KUKA KRL program: MyProgram_240().src

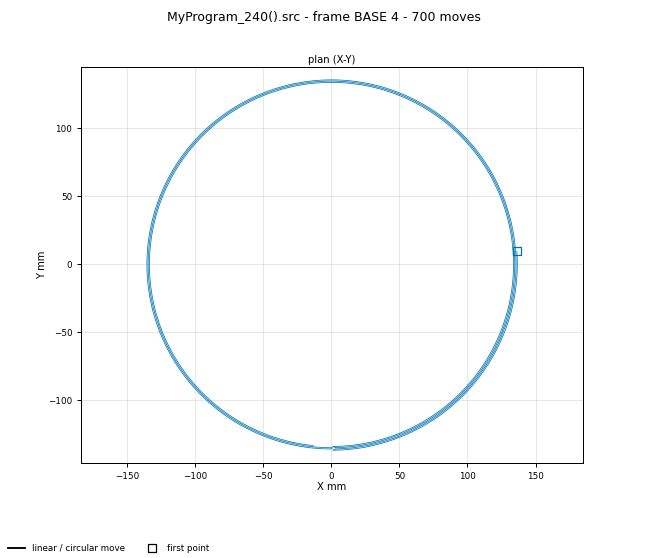
[picture p0: tool path of MyProgram_240().src in frame BASE 4, 700 of 700 moves have a stored position in this frame; points joined in program order, loops and branches not executed]
&ACCESS RVP
&REL 1
&PARAM TEMPLATE = C:\KRC\Roboter\Template\vorgabe
&PARAM EDITMASK = *
DEF MyProgram_240()
; ---- Setting reference (Base) ----
$BASE = BASE_DATA[4]

; --------------------------
; ---- Setting tool (TCP) ----
$TOOL = TOOL_DATA[3]
; --------------------------

$VEL.CP = VEL_APROX_PRINT
Startdeposition()
$VEL.CP = VEL_PRINT
LIN {X 136.2773,Y 9.5637,Z 161,A 0.3979,B 23.0272,C -1.0447,E1 23.2091,E2 806.9336} C_DIS
LIN {X 136.5182,Y 5.0682,Z 161,A -1.0464,B 23.0264,C -1.0618,E1 23.2093,E2 808.325} C_DIS
LIN {X 136.6137,Y -0.1543,Z 161,A -3.2724,B 23.0268,C -1.0528,E1 23.2093,E2 810.5594} C_DIS
LIN {X 136.5514,Y -4.0769,Z 161,A -4.8375,B 23.0268,C -1.0517,E1 23.2093,E2 812.1172} C_DIS
LIN {X 136.345,Y -8.5376,Z 161,A -6.6605,B 23.027,C -1.0482,E1 23.209,E2 813.9371} C_DIS
LIN {X 136.0456,Y -12.4414,Z 161,A -8.3456,B 23.0274,C -1.0406,E1 23.2086,E2 815.6307} C_DIS
LIN {X 135.6641,Y -16.0648,Z 161,A -10.3586,B 23.0286,C -1.0102,E1 23.2079,E2 817.7078} C_DIS
LIN {X 135.0038,Y -20.8989,Z 161,A -11.8021,B 23.0276,C -1.0351,E1 23.2074,E2 819.0787} C_DIS
LIN {X 134.4014,Y -24.4787,Z 161,A -13.4389,B 23.0281,C -1.0242,E1 23.2066,E2 820.7328} C_DIS
LIN {X 133.5686,Y -28.6745,Z 161,A -15.1069,B 23.0281,C -1.025,E1 23.2056,E2 822.388} C_DIS
LIN {X 132.7943,Y -32.0691,Z 161,A -16.5169,B 23.0281,C -1.023,E1 23.2047,E2 823.7942} C_DIS
LIN {X 131.9632,Y -35.3339,Z 161,A -17.9644,B 23.0284,C -1.0166,E1 23.2037,E2 825.2487} C_DIS
LIN {X 130.9854,Y -38.8039,Z 161,A -19.4634,B 23.0285,C -1.0125,E1 23.2025,E2 826.7489} C_DIS
LIN {X 129.5513,Y -43.3501,Z 161,A -21.4628,B 23.0288,C -1.0062,E1 23.2008,E2 828.7519} C_DIS
LIN {X 128.1195,Y -47.4171,Z 161,A -23.8257,B 23.0302,C -0.9715,E1 23.1985,E2 831.1885} C_DIS
LIN {X 126.3141,Y -52.0373,Z 161,A -25.224,B 23.029,C -1.0007,E1 23.1971,E2 832.504} C_DIS
LIN {X 124.3025,Y -56.6756,Z 161,A -27.3549,B 23.0293,C -0.9937,E1 23.1947,E2 834.6401} C_DIS
LIN {X 123.0552,Y -59.3326,Z 161,A -28.6015,B 23.0295,C -0.9891,E1 23.1932,E2 835.8908} C_DIS
LIN {X 121.4701,Y -62.5145,Z 161,A -30.119,B 23.0297,C -0.9833,E1 23.1913,E2 837.4144} C_DIS
LIN {X 119.0587,Y -66.9945,Z 161,A -32.2949,B 23.0301,C -0.9747,E1 23.1884,E2 839.5996} C_DIS
LIN {X 116.8471,Y -70.7814,Z 161,A -34.3743,B 23.0308,C -0.9568,E1 23.1853,E2 841.7128} C_DIS
LIN {X 115.0222,Y -73.7098,Z 161,A -35.319,B 23.0299,C -0.979,E1 23.184,E2 842.596} C_DIS
LIN {X 112.7004,Y -77.2131,Z 161,A -37.1335,B 23.0302,C -0.9713,E1 23.1812,E2 844.4202} C_DIS
LIN {X 110.946,Y -79.7139,Z 161,A -38.6151,B 23.0308,C -0.9572,E1 23.1788,E2 845.9297} C_DIS
LIN {X 108.2978,Y -83.2762,Z 161,A -40.4743,B 23.031,C -0.9523,E1 23.1756,E2 847.7917} C_DIS
LIN {X 105.5105,Y -86.7809,Z 161,A -42.2839,B 23.031,C -0.9508,E1 23.1724,E2 849.5958} C_DIS
LIN {X 102.8746,Y -89.8891,Z 161,A -44.0205,B 23.0313,C -0.945,E1 23.1693,E2 851.3386} C_DIS
LIN {X 100.0782,Y -92.9925,Z 161,A -45.7792,B 23.0314,C -0.9401,E1 23.166,E2 853.1011} C_DIS
LIN {X 96.8908,Y -96.3089,Z 161,A -47.6911,B 23.0316,C -0.9363,E1 23.1622,E2 855.0138} C_DIS
LIN {X 93.7473,Y -99.3714,Z 161,A -49.4881,B 23.0316,C -0.9341,E1 23.1586,E2 856.8082} C_DIS
LIN {X 90.5239,Y -102.3164,Z 161,A -51.3153,B 23.0318,C -0.93,E1 23.1548,E2 858.6377} C_DIS
LIN {X 87.2594,Y -105.1145,Z 161,A -53.1447,B 23.032,C -0.9246,E1 23.1509,E2 860.4732} C_DIS
LIN {X 83.7135,Y -107.9596,Z 161,A -55.0296,B 23.0322,C -0.9216,E1 23.1468,E2 862.3582} C_DIS
LIN {X 79.9438,Y -110.7803,Z 161,A -56.981,B 23.0322,C -0.9186,E1 23.1424,E2 864.3095} C_DIS
LIN {X 76.3648,Y -113.2771,Z 161,A -58.824,B 23.0324,C -0.9142,E1 23.1381,E2 866.1567} C_DIS
LIN {X 72.5813,Y -115.7382,Z 161,A -60.7513,B 23.0326,C -0.9088,E1 23.1336,E2 868.0909} C_DIS
LIN {X 68.7664,Y -118.0447,Z 161,A -62.5822,B 23.0326,C -0.9074,E1 23.1292,E2 869.9194} C_DIS
LIN {X 64.8661,Y -120.2317,Z 161,A -64.9487,B 23.0337,C -0.879,E1 23.1232,E2 872.3506} C_DIS
LIN {X 60.5233,Y -122.4729,Z 161,A -66.0976,B 23.0322,C -0.9217,E1 23.1207,E2 873.3874} C_DIS
LIN {X 58.242,Y -123.5762,Z 161,A -67.4262,B 23.0327,C -0.9063,E1 23.1172,E2 874.7514} C_DIS
LIN {X 54.9164,Y -125.0898,Z 161,A -69.3172,B 23.0335,C -0.8857,E1 23.1122,E2 876.6899} C_DIS
LIN {X 51.6442,Y -126.4751,Z 161,A -70.416,B 23.0328,C -0.9034,E1 23.1095,E2 877.7406} C_DIS
LIN {X 45.2029,Y -128.9172,Z 161,A -73.1919,B 23.0328,C -0.9053,E1 23.1023,E2 880.5052} C_DIS
LIN {X 41.5898,Y -130.1269,Z 161,A -74.9321,B 23.0331,C -0.8961,E1 23.0976,E2 882.2652} C_DIS
LIN {X 36.528,Y -131.6378,Z 161,A -77.0528,B 23.0331,C -0.8984,E1 23.092,E2 884.3759} C_DIS
LIN {X 33.7209,Y -132.3845,Z 161,A -78.3762,B 23.0333,C -0.8919,E1 23.0884,E2 885.714} C_DIS
LIN {X 30.5077,Y -133.1617,Z 161,A -79.7785,B 23.0333,C -0.8897,E1 23.0845,E2 887.1194} C_DIS
LIN {X 26.5179,Y -134.0153,Z 161,A -81.6868,B 23.0338,C -0.8783,E1 23.0792,E2 889.0544} C_DIS
LIN {X 22.9609,Y -134.6693,Z 161,A -82.9925,B 23.0334,C -0.8877,E1 23.0757,E2 890.3344} C_DIS
LIN {X 19.4058,Y -135.2265,Z 161,A -84.8817,B 23.0341,C -0.8677,E1 23.0704,E2 892.2729} C_DIS
LIN {X 15.342,Y -135.7496,Z 161,A -86.2543,B 23.0336,C -0.8839,E1 23.0667,E2 893.6031} C_DIS
LIN {X 8.2701,Y -136.3615,Z 161,A -89.1847,B 23.0336,C -0.8848,E1 23.0585,E2 896.5294} C_DIS
LIN {X 0.9864,Y -136.6083,Z 161,A -93.055,B 23.035,C -0.8438,E1 23.0474,E2 900.5038} C_DIS
Enddeposition()
LIN {X 0.9864,Y -136.6083,Z 161,A -93.055,B 23.035,C -0.8438,E1 23.0474,E2 900.5038} C_DIS
Startdeposition()
$VEL.CP = VEL_PRINT
LIN {X 2.6306,Y -135.6628,Z 161,A -90.3615,B 21.7658,C -0.7295,E1 21.7824,E2 897.9751} C_DIS
LIN {X 6.721,Y -135.5212,Z 161,A -88.7348,B 21.766,C -0.7253,E1 21.7869,E2 896.3603} C_DIS
LIN {X 9.445,Y -135.3593,Z 161,A -87.4479,B 21.7658,C -0.7322,E1 21.7905,E2 895.0556} C_DIS
LIN {X 14.134,Y -134.9501,Z 161,A -85.5629,B 21.7658,C -0.7283,E1 21.7957,E2 893.1824} C_DIS
LIN {X 18.0786,Y -134.4786,Z 161,A -83.8012,B 21.7658,C -0.7334,E1 21.8006,E2 891.4087} C_DIS
LIN {X 22.3172,Y -133.8397,Z 161,A -82.1872,B 21.766,C -0.7253,E1 21.805,E2 889.8183} C_DIS
LIN {X 24.8651,Y -133.3913,Z 161,A -80.9711,B 21.7658,C -0.732,E1 21.8084,E2 888.5856} C_DIS
LIN {X 28.3569,Y -132.6916,Z 161,A -79.5518,B 21.7658,C -0.7293,E1 21.8122,E2 887.1758} C_DIS
LIN {X 31.5596,Y -131.9665,Z 161,A -78.1631,B 21.7658,C -0.7307,E1 21.816,E2 885.7857} C_DIS
LIN {X 34.2506,Y -131.2956,Z 161,A -76.8928,B 21.7656,C -0.7366,E1 21.8195,E2 884.5017} C_DIS
LIN {X 40.5935,Y -129.4745,Z 161,A -74.0549,B 21.7654,C -0.7422,E1 21.8271,E2 881.6545} C_DIS
LIN {X 44.4809,Y -128.1894,Z 161,A -72.4077,B 21.7654,C -0.7404,E1 21.8314,E2 880.016} C_DIS
LIN {X 48.4743,Y -126.7353,Z 161,A -70.6142,B 21.7654,C -0.7426,E1 21.8361,E2 878.2208} C_DIS
LIN {X 52.0834,Y -125.2933,Z 161,A -68.9248,B 21.7653,C -0.7473,E1 21.8405,E2 876.5234} C_DIS
LIN {X 56.601,Y -123.3187,Z 161,A -67.1132,B 21.7656,C -0.7373,E1 21.8451,E2 874.7439} C_DIS
LIN {X 60.0155,Y -121.6929,Z 161,A -64.3194,B 21.7635,C -0.7986,E1 21.8525,E2 871.7941} C_DIS
LIN {X 66.7124,Y -118.157,Z 161,A -62.0959,B 21.765,C -0.756,E1 21.8576,E2 869.6927} C_DIS
LIN {X 72.0742,Y -114.9654,Z 161,A -59.4888,B 21.7649,C -0.7595,E1 21.8638,E2 867.0857} C_DIS
LIN {X 75.5582,Y -112.7058,Z 161,A -57.7533,B 21.7648,C -0.762,E1 21.8679,E2 865.3501} C_DIS
LIN {X 79.2761,Y -110.1229,Z 161,A -55.828,B 21.7646,C -0.7665,E1 21.8722,E2 863.4205} C_DIS
LIN {X 82.83,Y -107.4751,Z 161,A -53.9837,B 21.7646,C -0.7692,E1 21.8763,E2 861.577} C_DIS
LIN {X 86.0296,Y -104.931,Z 161,A -52.2698,B 21.7644,C -0.7723,E1 21.8801,E2 859.8621} C_DIS
LIN {X 89.4999,Y -101.9876,Z 161,A -50.3307,B 21.7643,C -0.7775,E1 21.8842,E2 857.918} C_DIS
LIN {X 92.7399,Y -99.0506,Z 161,A -48.5154,B 21.7642,C -0.7803,E1 21.8879,E2 856.1039} C_DIS
LIN {X 95.8163,Y -96.0774,Z 161,A -46.7327,B 21.7641,C -0.7834,E1 21.8915,E2 854.3216} C_DIS
LIN {X 98.8991,Y -92.9011,Z 161,A -44.8508,B 21.7639,C -0.7886,E1 21.8951,E2 852.4351} C_DIS
LIN {X 101.9435,Y -89.5503,Z 161,A -42.9731,B 21.7638,C -0.7918,E1 21.8986,E2 850.5587} C_DIS
LIN {X 104.6052,Y -86.4253,Z 161,A -41.2947,B 21.7638,C -0.7936,E1 21.9016,E2 848.8846} C_DIS
LIN {X 107.2944,Y -83.0631,Z 161,A -39.44,B 21.7635,C -0.8002,E1 21.9048,E2 847.0222} C_DIS
LIN {X 110.0674,Y -79.3526,Z 161,A -37.6745,B 21.7636,C -0.796,E1 21.9077,E2 845.2779} C_DIS
LIN {X 113.15,Y -74.8916,Z 161,A -35.3067,B 21.7633,C -0.8062,E1 21.9115,E2 842.8963} C_DIS
LIN {X 116.0911,Y -70.2454,Z 161,A -32.9144,B 21.7629,C -0.8163,E1 21.915,E2 840.4912} C_DIS
LIN {X 117.6865,Y -67.5395,Z 161,A -31.2671,B 21.7622,C -0.8362,E1 21.9174,E2 838.8005} C_DIS
LIN {X 119.6001,Y -64.089,Z 161,A -29.8843,B 21.7625,C -0.8268,E1 21.9191,E2 837.4512} C_DIS
LIN {X 121.5521,Y -60.301,Z 161,A -28.2528,B 21.7626,C -0.8238,E1 21.9212,E2 835.8381} C_DIS
LIN {X 122.9704,Y -57.3542,Z 161,A -27.0274,B 21.7628,C -0.8201,E1 21.9226,E2 834.63} C_DIS
LIN {X 124.2951,Y -54.4258,Z 161,A -25.4063,B 21.7621,C -0.8374,E1 21.9245,E2 832.973} C_DIS
LIN {X 127.902,Y -45.3069,Z 161,A -21.4308,B 21.762,C -0.8417,E1 21.9285,E2 829.0118} C_DIS
LIN {X 129.6738,Y -39.9479,Z 161,A -19.1656,B 21.762,C -0.8432,E1 21.9304,E2 826.7574} C_DIS
LIN {X 130.6686,Y -36.5623,Z 161,A -17.5786,B 21.7616,C -0.8527,E1 21.9317,E2 825.1555} C_DIS
LIN {X 131.5001,Y -33.4486,Z 161,A -16.2258,B 21.7614,C -0.8566,E1 21.9326,E2 823.8013} C_DIS
LIN {X 132.3825,Y -29.7689,Z 161,A -14.5067,B 21.761,C -0.8678,E1 21.9337,E2 822.064} C_DIS
LIN {X 133.3015,Y -25.3348,Z 161,A -12.6917,B 21.761,C -0.869,E1 21.9347,E2 820.2581} C_DIS
LIN {X 134.0395,Y -21.0869,Z 161,A -11.1256,B 21.7612,C -0.8621,E1 21.9354,E2 818.7212} C_DIS
LIN {X 134.4989,Y -17.9238,Z 161,A -9.451,B 21.7604,C -0.8827,E1 21.9361,E2 817.003} C_DIS
LIN {X 135.0397,Y -13.2483,Z 161,A -7.7651,B 21.7608,C -0.8739,E1 21.9366,E2 815.3521} C_DIS
LIN {X 135.317,Y -10.025,Z 161,A -6.2881,B 21.7604,C -0.8839,E1 21.9369,E2 813.8587} C_DIS
LIN {X 135.5188,Y -6.7689,Z 161,A -4.8555,B 21.7601,C -0.8911,E1 21.9371,E2 812.4167} C_DIS
LIN {X 135.6615,Y -2.7083,Z 161,A -3.0725,B 21.7598,C -0.9,E1 21.9372,E2 810.6223} C_DIS
LIN {X 135.6756,Y 1.8649,Z 161,A -1.2349,B 21.7598,C -0.9015,E1 21.9372,E2 808.7933} C_DIS
LIN {X 135.5773,Y 5.478,Z 161,A 0.0506,B 21.76,C -0.8943,E1 21.9372,E2 807.5359} C_DIS
LIN {X 135.424,Y 8.4577,Z 161,A 1.4958,B 21.7595,C -0.9076,E1 21.9369,E2 806.0652} C_DIS
LIN {X 135.1194,Y 12.4177,Z 161,A 3.254,B 21.7591,C -0.917,E1 21.9365,E2 804.2939} C_DIS
LIN {X 134.6789,Y 16.5206,Z 161,A 5.014,B 21.7588,C -0.9234,E1 21.9359,E2 802.5289} C_DIS
LIN {X 134.157,Y 20.3276,Z 161,A 6.5505,B 21.7588,C -0.9242,E1 21.9353,E2 801.0008} C_DIS
LIN {X 133.5954,Y 23.7364,Z 161,A 7.9477,B 21.7588,C -0.9257,E1 21.9346,E2 799.6092} C_DIS
LIN {X 132.9372,Y 27.1812,Z 161,A 9.4648,B 21.7585,C -0.9322,E1 21.9338,E2 798.0852} C_DIS
LIN {X 131.9188,Y 31.7572,Z 161,A 11.3888,B 21.7583,C -0.9355,E1 21.9326,E2 796.1652} C_DIS
LIN {X 130.9966,Y 35.3717,Z 161,A 13.0456,B 21.758,C -0.9444,E1 21.9314,E2 794.4958} C_DIS
LIN {X 127.8094,Y 45.5637,Z 161,A 17.4828,B 21.7576,C -0.9542,E1 21.9276,E2 790.0616} C_DIS
LIN {X 125.7762,Y 50.9062,Z 161,A 19.7346,B 21.7576,C -0.9532,E1 21.9254,E2 787.8269} C_DIS
LIN {X 124.6706,Y 53.5573,Z 161,A 21.0157,B 21.7573,C -0.9601,E1 21.9239,E2 786.5356} C_DIS
LIN {X 123.2293,Y 56.7944,Z 161,A 22.3641,B 21.7574,C -0.9571,E1 21.9224,E2 785.2039} C_DIS
LIN {X 121.8558,Y 59.6853,Z 161,A 23.906,B 21.7569,C -0.9703,E1 21.9205,E2 783.6363} C_DIS
LIN {X 120.1715,Y 63.0066,Z 161,A 25.3923,B 21.7569,C -0.9703,E1 21.9186,E2 782.1589} C_DIS
LIN {X 118.0968,Y 66.8196,Z 161,A 27.3535,B 21.7564,C -0.9817,E1 21.9159,E2 780.1793} C_DIS
LIN {X 115.9673,Y 70.4502,Z 161,A 29.0848,B 21.7564,C -0.9841,E1 21.9135,E2 778.4518} C_DIS
LIN {X 113.606,Y 74.1983,Z 161,A 30.9425,B 21.7561,C -0.9884,E1 21.9107,E2 776.5935} C_DIS
LIN {X 111.8562,Y 76.8098,Z 161,A 32.7606,B 21.7549,C -1.016,E1 21.9077,E2 774.7118} C_DIS
LIN {X 109.0292,Y 80.7731,Z 161,A 34.3198,B 21.7558,C -0.9966,E1 21.9052,E2 773.2134} C_DIS
LIN {X 105.9568,Y 84.7633,Z 161,A 36.4456,B 21.7555,C -1.0017,E1 21.9015,E2 771.0856} C_DIS
LIN {X 103.0638,Y 88.2586,Z 161,A 38.231,B 21.7556,C -0.9998,E1 21.8983,E2 769.3149} C_DIS
LIN {X 99.7809,Y 91.9528,Z 161,A 40.3381,B 21.7554,C -1.0055,E1 21.8944,E2 767.2033} C_DIS
LIN {X 96.9434,Y 94.9397,Z 161,A 42.1274,B 21.7551,C -1.0117,E1 21.8909,E2 765.4063} C_DIS
LIN {X 94.8714,Y 97.0104,Z 161,A 43.4385,B 21.7548,C -1.018,E1 21.8883,E2 764.0849} C_DIS
LIN {X 91.3906,Y 100.2966,Z 161,A 45.411,B 21.7548,C -1.0197,E1 21.8843,E2 762.117} C_DIS
LIN {X 88.4188,Y 102.9257,Z 161,A 48.0168,B 21.7525,C -1.0685,E1 21.8785,E2 759.392} C_DIS
LIN {X 82.6709,Y 107.5973,Z 161,A 50.1675,B 21.7544,C -1.0265,E1 21.874,E2 757.3633} C_DIS
LIN {X 78.7472,Y 110.5011,Z 161,A 52.2253,B 21.7543,C -1.03,E1 21.8694,E2 755.3048} C_DIS
LIN {X 75.2259,Y 112.9276,Z 161,A 54.0074,B 21.7542,C -1.0319,E1 21.8652,E2 753.5247} C_DIS
LIN {X 71.3591,Y 115.4105,Z 161,A 55.926,B 21.7542,C -1.0338,E1 21.8607,E2 751.608} C_DIS
LIN {X 67.6548,Y 117.6203,Z 161,A 57.7882,B 21.7539,C -1.0385,E1 21.8562,E2 749.7399} C_DIS
LIN {X 63.7967,Y 119.7566,Z 161,A 59.6822,B 21.7537,C -1.0426,E1 21.8515,E2 747.8413} C_DIS
LIN {X 60.4556,Y 121.4758,Z 161,A 61.1704,B 21.7538,C -1.04,E1 21.8479,E2 746.3649} C_DIS
LIN {X 57.2122,Y 123.0361,Z 161,A 62.6232,B 21.7538,C -1.0386,E1 21.8442,E2 744.92} C_DIS
LIN {X 53.899,Y 124.5229,Z 161,A 64.1049,B 21.7539,C -1.0379,E1 21.8404,E2 743.4443} C_DIS
LIN {X 46.6483,Y 127.4184,Z 161,A 67.3702,B 21.7539,C -1.0397,E1 21.832,E2 740.1828} C_DIS
LIN {X 42.5099,Y 128.857,Z 161,A 69.3414,B 21.7535,C -1.047,E1 21.8267,E2 738.1963} C_DIS
LIN {X 38.5045,Y 130.1101,Z 161,A 71.0992,B 21.7535,C -1.0477,E1 21.822,E2 736.4403} C_DIS
LIN {X 35.0814,Y 131.074,Z 161,A 72.5366,B 21.7535,C -1.0458,E1 21.8182,E2 735.0109} C_DIS
LIN {X 31.831,Y 131.901,Z 161,A 73.8763,B 21.7537,C -1.0431,E1 21.8146,E2 733.6809} C_DIS
LIN {X 28.7421,Y 132.6085,Z 161,A 75.383,B 21.7533,C -1.0517,E1 21.8104,E2 732.1534} C_DIS
LIN {X 24.7943,Y 133.4048,Z 161,A 76.9366,B 21.7536,C -1.0455,E1 21.8062,E2 730.6184} C_DIS
LIN {X 20.8451,Y 134.0769,Z 161,A 78.478,B 21.7539,C -1.0392,E1 21.802,E2 729.096} C_DIS
LIN {X 18.6136,Y 134.4061,Z 161,A 79.7449,B 21.7532,C -1.054,E1 21.7984,E2 727.7904} C_DIS
LIN {X 14.7979,Y 134.8786,Z 161,A 81.3068,B 21.7532,C -1.0515,E1 21.7941,E2 726.2366} C_DIS
LIN {X 11.9597,Y 135.1607,Z 161,A 82.5203,B 21.7532,C -1.0521,E1 21.7907,E2 725.0224} C_DIS
LIN {X 7.7951,Y 135.4648,Z 161,A 84.3117,B 21.7532,C -1.0535,E1 21.7857,E2 723.2282} C_DIS
LIN {X 3.449,Y 135.6443,Z 161,A 86.2031,B 21.7531,C -1.0559,E1 21.7804,E2 721.3308} C_DIS
LIN {X -0.0735,Y 135.6895,Z 161,A 87.6782,B 21.7531,C -1.0551,E1 21.7763,E2 719.858} C_DIS
LIN {X -4.1066,Y 135.6261,Z 161,A 89.3542,B 21.7532,C -1.0534,E1 21.7716,E2 718.1863} C_DIS
LIN {X -8.3893,Y 135.4282,Z 161,A 91.1318,B 21.7533,C -1.0513,E1 21.7667,E2 716.4138} C_DIS
LIN {X -12.9086,Y 135.0723,Z 161,A 92.8361,B 21.7538,C -1.0409,E1 21.762,E2 714.7366} C_DIS
LIN {X -15.9106,Y 134.7517,Z 161,A 94.0719,B 21.7538,C -1.0385,E1 21.7586,E2 713.5065} C_DIS
LIN {X -19.1715,Y 134.3264,Z 161,A 95.6577,B 21.7535,C -1.0466,E1 21.7542,E2 711.8974} C_DIS
LIN {X -22.7522,Y 133.7671,Z 161,A 97.2253,B 21.7535,C -1.0472,E1 21.7498,E2 710.3264} C_DIS
LIN {X -26.7692,Y 133.0211,Z 161,A 98.8877,B 21.7537,C -1.0431,E1 21.7453,E2 708.6731} C_DIS
LIN {X -30.0117,Y 132.327,Z 161,A 100.3431,B 21.7537,C -1.0444,E1 21.7413,E2 707.212} C_DIS
LIN {X -33.3937,Y 131.5141,Z 161,A 101.8139,B 21.7537,C -1.0431,E1 21.7373,E2 705.7422} C_DIS
LIN {X -41.2355,Y 129.2699,Z 161,A 105.3327,B 21.7537,C -1.0428,E1 21.7279,E2 702.2177} C_DIS
LIN {X -44.9986,Y 128.0099,Z 161,A 107.0495,B 21.7537,C -1.0426,E1 21.7233,E2 700.4975} C_DIS
LIN {X -48.5735,Y 126.6967,Z 161,A 108.4612,B 21.7542,C -1.0317,E1 21.7197,E2 699.1118} C_DIS
LIN {X -51.8102,Y 125.4074,Z 161,A 109.8953,B 21.7544,C -1.0281,E1 21.716,E2 697.6838} C_DIS
LIN {X -54.485,Y 124.2695,Z 161,A 111.3741,B 21.7539,C -1.0375,E1 21.7122,E2 696.1754} C_DIS
LIN {X -58.2306,Y 122.5574,Z 161,A 112.7848,B 21.7547,C -1.0203,E1 21.7087,E2 694.8071} C_DIS
LIN {X -61.2691,Y 121.067,Z 161,A 114.5593,B 21.7541,C -1.0334,E1 21.7042,E2 692.9918} C_DIS
LIN {X -66.3889,Y 118.3389,Z 161,A 117.0044,B 21.7543,C -1.0291,E1 21.6982,E2 690.5503} C_DIS
LIN {X -70.5015,Y 115.9363,Z 161,A 118.9693,B 21.7546,C -1.0234,E1 21.6935,E2 688.5937} C_DIS
LIN {X -74.8528,Y 113.1755,Z 161,A 121.8836,B 21.7533,C -1.0521,E1 21.6865,E2 685.5906} C_DIS
LIN {X -79.6697,Y 109.8376,Z 161,A 123.6709,B 21.7549,C -1.0166,E1 21.6826,E2 683.8922} C_DIS
LIN {X -82.3618,Y 107.8337,Z 161,A 125.4147,B 21.7544,C -1.0281,E1 21.6787,E2 682.11} C_DIS
LIN {X -85.4101,Y 105.4361,Z 161,A 126.7086,B 21.7552,C -1.0095,E1 21.6759,E2 680.8609} C_DIS
LIN {X -88.7115,Y 102.6737,Z 161,A 128.5803,B 21.7552,C -1.0078,E1 21.6719,E2 678.9852} C_DIS
LIN {X -92.1214,Y 99.6261,Z 161,A 130.5442,B 21.7554,C -1.0048,E1 21.6679,E2 677.0201} C_DIS
LIN {X -95.2819,Y 96.6077,Z 161,A 132.3637,B 21.7556,C -0.9994,E1 21.6642,E2 675.2066} C_DIS
LIN {X -98.1476,Y 93.6943,Z 161,A 134.044,B 21.7559,C -0.9932,E1 21.661,E2 673.5345} C_DIS
LIN {X -100.9175,Y 90.7044,Z 161,A 135.8256,B 21.7559,C -0.9916,E1 21.6576,E2 671.7481} C_DIS
LIN {X -105.2895,Y 85.5906,Z 161,A 138.6205,B 21.7564,C -0.9823,E1 21.6526,E2 668.9635} C_DIS
LIN {X -108.6887,Y 81.2305,Z 161,A 141.0706,B 21.7564,C -0.9811,E1 21.6485,E2 666.5029} C_DIS
LIN {X -110.9298,Y 78.1419,Z 161,A 143.0908,B 21.7559,C -0.9945,E1 21.6451,E2 664.4348} C_DIS
LIN {X -113.4209,Y 74.4801,Z 161,A 144.4907,B 21.757,C -0.9689,E1 21.6431,E2 663.0962} C_DIS
LIN {X -115.6634,Y 70.9475,Z 161,A 146.2696,B 21.7571,C -0.9645,E1 21.6404,E2 661.3188} C_DIS
LIN {X -117.6966,Y 67.5217,Z 161,A 147.7352,B 21.7577,C -0.9503,E1 21.6384,E2 659.8827} C_DIS
LIN {X -119.9419,Y 63.4439,Z 161,A 149.8673,B 21.7577,C -0.9518,E1 21.6355,E2 657.7335} C_DIS
LIN {X -121.4837,Y 60.4397,Z 161,A 151.5472,B 21.7574,C -0.9586,E1 21.6334,E2 656.0247} C_DIS
LIN {X -123.6736,Y 55.822,Z 161,A 153.5716,B 21.7579,C -0.9464,E1 21.631,E2 654.0205} C_DIS
LIN {X -125.1307,Y 52.4727,Z 161,A 155.0695,B 21.7582,C -0.9398,E1 21.6294,E2 652.5307} C_DIS
LIN {X -126.2395,Y 49.7498,Z 161,A 156.4219,B 21.7582,C -0.9408,E1 21.628,E2 651.1669} C_DIS
LIN {X -127.5477,Y 46.2895,Z 161,A 157.8668,B 21.7585,C -0.931,E1 21.6266,E2 649.739} C_DIS
LIN {X -128.5417,Y 43.4566,Z 161,A 159.3197,B 21.7584,C -0.935,E1 21.6253,E2 648.2656} C_DIS
LIN {X -129.6308,Y 40.0885,Z 161,A 160.711,B 21.7587,C -0.9259,E1 21.6241,E2 646.8896} C_DIS
LIN {X -130.6087,Y 36.7763,Z 161,A 162.1278,B 21.759,C -0.9196,E1 21.623,E2 645.4805} C_DIS
LIN {X -131.4745,Y 33.5498,Z 161,A 163.5569,B 21.7591,C -0.9159,E1 21.622,E2 644.0515} C_DIS
LIN {X -132.2559,Y 30.3232,Z 161,A 164.9557,B 21.7593,C -0.9114,E1 21.6211,E2 642.6555} C_DIS
LIN {X -132.8535,Y 27.5927,Z 161,A 166.2341,B 21.7593,C -0.9118,E1 21.6204,E2 641.3671} C_DIS
LIN {X -133.507,Y 24.2301,Z 161,A 167.4819,B 21.7598,C -0.8987,E1 21.6197,E2 640.1462} C_DIS
LIN {X -134.0793,Y 20.8299,Z 161,A 169.1016,B 21.7598,C -0.9011,E1 21.619,E2 638.5089} C_DIS
LIN {X -134.5669,Y 17.4053,Z 161,A 170.6261,B 21.7598,C -0.8991,E1 21.6184,E2 636.979} C_DIS
LIN {X -135.0616,Y 13.0198,Z 161,A 172.4817,B 21.76,C -0.8928,E1 21.6179,E2 635.1276} C_DIS
LIN {X -135.4054,Y 8.7594,Z 161,A 174.3182,B 21.7602,C -0.8884,E1 21.6175,E2 633.2902} C_DIS
LIN {X -135.5926,Y 5.0854,Z 161,A 175.8945,B 21.7604,C -0.8844,E1 21.6173,E2 631.7137} C_DIS
LIN {X -135.6855,Y 0.8916,Z 161,A 177.628,B 21.7607,C -0.8771,E1 21.6173,E2 629.9879} C_DIS
LIN {X -135.659,Y -2.862,Z 161,A 179.3405,B 21.7607,C -0.8775,E1 21.6173,E2 628.2622} C_DIS
LIN {X -135.5073,Y -6.9975,Z 161,A -179.0048,B 21.761,C -0.8679,E1 21.6175,E2 626.6218} C_DIS
LIN {X -135.232,Y -11.116,Z 161,A -177.2662,B 21.7612,C -0.8622,E1 21.6179,E2 624.8867} C_DIS
LIN {X -134.9048,Y -14.5547,Z 161,A -175.8003,B 21.7614,C -0.8579,E1 21.6183,E2 623.4221} C_DIS
LIN {X -134.431,Y -18.4399,Z 161,A -174.0261,B 21.7614,C -0.8579,E1 21.6189,E2 621.6356} C_DIS
LIN {X -133.8734,Y -22.1149,Z 161,A -172.55,B 21.7617,C -0.8489,E1 21.6196,E2 620.1735} C_DIS
LIN {X -133.3708,Y -24.9719,Z 161,A -171.4418,B 21.762,C -0.8401,E1 21.6201,E2 619.0817} C_DIS
LIN {X -132.1859,Y -30.6296,Z 161,A -168.7455,B 21.762,C -0.8435,E1 21.6218,E2 616.3575} C_DIS
LIN {X -131.2802,Y -34.3081,Z 161,A -166.9877,B 21.7618,C -0.8454,E1 21.623,E2 614.5824} C_DIS
LIN {X -129.8793,Y -39.2766,Z 161,A -165.0969,B 21.7625,C -0.8263,E1 21.6244,E2 612.7307} C_DIS
LIN {X -129.0208,Y -42.0153,Z 161,A -163.6523,B 21.7623,C -0.8328,E1 21.6257,E2 611.259} C_DIS
LIN {X -127.7402,Y -45.7555,Z 161,A -162.3613,B 21.7631,C -0.8115,E1 21.6268,E2 610.0172} C_DIS
LIN {X -126.632,Y -48.7402,Z 161,A -160.7495,B 21.7628,C -0.8191,E1 21.6284,E2 608.3741} C_DIS
LIN {X -125.2904,Y -52.0903,Z 161,A -159.2589,B 21.763,C -0.8132,E1 21.63,E2 606.8898} C_DIS
LIN {X -124.1683,Y -54.716,Z 161,A -157.4205,B 21.7621,C -0.8374,E1 21.6322,E2 604.9738} C_DIS
LIN {X -122.0569,Y -59.2777,Z 161,A -155.912,B 21.7633,C -0.8045,E1 21.6339,E2 603.545} C_DIS
LIN {X -120.6041,Y -62.1785,Z 161,A -154.3801,B 21.7633,C -0.8078,E1 21.6359,E2 601.9946} C_DIS
LIN {X -118.3545,Y -66.3612,Z 161,A -152.4228,B 21.7635,C -0.8003,E1 21.6385,E2 600.0458} C_DIS
LIN {X -116.2025,Y -70.0612,Z 161,A -150.5815,B 21.7635,C -0.7969,E1 21.6411,E2 598.2024} C_DIS
LIN {X -113.7867,Y -73.9199,Z 161,A -148.7475,B 21.7639,C -0.7881,E1 21.6438,E2 596.3816} C_DIS
LIN {X -111.3799,Y -77.4989,Z 161,A -146.8885,B 21.7639,C -0.7851,E1 21.6468,E2 594.5199} C_DIS
LIN {X -109.0213,Y -80.7838,Z 161,A -145.1275,B 21.7641,C -0.7832,E1 21.6497,E2 592.754} C_DIS
LIN {X -106.4705,Y -84.1175,Z 161,A -143.3363,B 21.7641,C -0.7798,E1 21.6528,E2 590.9623} C_DIS
LIN {X -103.6739,Y -87.5412,Z 161,A -141.3776,B 21.7641,C -0.7795,E1 21.6563,E2 588.9939} C_DIS
LIN {X -100.4244,Y -91.2498,Z 161,A -139.3546,B 21.7644,C -0.7721,E1 21.66,E2 586.9802} C_DIS
LIN {X -97.3609,Y -94.5117,Z 161,A -137.6966,B 21.7649,C -0.7577,E1 21.6632,E2 585.3528} C_DIS
LIN {X -95.0347,Y -96.8502,Z 161,A -136.0886,B 21.7647,C -0.7643,E1 21.6664,E2 583.719} C_DIS
LIN {X -91.9812,Y -99.755,Z 161,A -134.2787,B 21.7647,C -0.762,E1 21.6701,E2 581.9067} C_DIS
LIN {X -87.3021,Y -103.8745,Z 161,A -131.6173,B 21.7649,C -0.7582,E1 21.6757,E2 579.2435} C_DIS
LIN {X -83.9274,Y -106.6198,Z 161,A -129.8066,B 21.7651,C -0.7536,E1 21.6796,E2 577.4374} C_DIS
LIN {X -80.6269,Y -109.1375,Z 161,A -127.9773,B 21.7651,C -0.754,E1 21.6838,E2 575.5995} C_DIS
LIN {X -77.0748,Y -111.6743,Z 161,A -126.1278,B 21.7651,C -0.7512,E1 21.688,E2 573.7502} C_DIS
LIN {X -74.0448,Y -113.7056,Z 161,A -124.265,B 21.7647,C -0.7633,E1 21.6924,E2 571.8474} C_DIS
LIN {X -70.5634,Y -115.8986,Z 161,A -122.8227,B 21.7653,C -0.7473,E1 21.6958,E2 570.4432} C_DIS
LIN {X -66.4685,Y -118.2942,Z 161,A -120.9182,B 21.7655,C -0.74,E1 21.7004,E2 568.552} C_DIS
LIN {X -63.6574,Y -119.8298,Z 161,A -119.4928,B 21.7655,C -0.7415,E1 21.7039,E2 567.1178} C_DIS
LIN {X -60.2545,Y -121.575,Z 161,A -117.9704,B 21.7657,C -0.7353,E1 21.7077,E2 565.6075} C_DIS
LIN {X -57.5053,Y -122.9006,Z 161,A -116.6289,B 21.7657,C -0.7361,E1 21.7111,E2 564.2597} C_DIS
LIN {X -54.7338,Y -124.1603,Z 161,A -114.7547,B 21.7648,C -0.7617,E1 21.7161,E2 562.3111} C_DIS
LIN {X -49.9472,Y -126.1627,Z 161,A -113.2112,B 21.7658,C -0.7297,E1 21.7198,E2 560.8503} C_DIS
LIN {X -45.3558,Y -127.8844,Z 161,A -110.9686,B 21.7656,C -0.7357,E1 21.7258,E2 558.5862} C_DIS
LIN {X -41.4162,Y -129.2122,Z 161,A -109.3781,B 21.7659,C -0.7267,E1 21.7299,E2 557.0165} C_DIS
LIN {X -38.36,Y -130.1524,Z 161,A -108.0279,B 21.7659,C -0.7257,E1 21.7335,E2 555.6664} C_DIS
LIN {X -35.0745,Y -131.0759,Z 161,A -106.6479,B 21.7661,C -0.7219,E1 21.7372,E2 554.2941} C_DIS
LIN {X -32.3609,Y -131.7733,Z 161,A -105.3058,B 21.7659,C -0.7286,E1 21.7409,E2 552.9318} C_DIS
LIN {X -28.5349,Y -132.6532,Z 161,A -103.8032,B 21.7661,C -0.7206,E1 21.745,E2 551.4485} C_DIS
LIN {X -23.5022,Y -133.6373,Z 161,A -101.5285,B 21.766,C -0.7248,E1 21.7513,E2 549.1597} C_DIS
LIN {X -19.2533,Y -134.3147,Z 161,A -99.7477,B 21.766,C -0.7226,E1 21.7562,E2 547.383} C_DIS
LIN {X -15.4289,Y -134.8092,Z 161,A -97.9709,B 21.7658,C -0.7292,E1 21.7611,E2 545.5869} C_DIS
LIN {X -9.4132,Y -135.3616,Z 161,A -95.4725,B 21.7659,C -0.7266,E1 21.7681,E2 543.0943} C_DIS
LIN {X -5.0542,Y -135.5938,Z 161,A -93.7426,B 21.7661,C -0.7214,E1 21.7729,E2 541.378} C_DIS
LIN {X -0.237,Y -135.6886,Z 161,A -91.462,B 21.7657,C -0.7333,E1 21.7793,E2 539.0652} C_DIS
LIN {X -0.237,Y -135.6886,Z 161,A -91.462,B 21.7657,C -0.7333,E1 21.7793,E2 539.0652} C_DIS
Enddeposition()
LIN {X 0.973,Y -134.7603,Z 161,A -91.2443,B 20.6491,C -0.5507,E1 20.6575,E2 539.2391} C_DIS
Startdeposition()
$VEL.CP = VEL_PRINT
LIN {X -1.314,Y -134.7584,Z 161,A -92.4001,B 20.6493,C -0.5425,E1 20.6542,E2 540.4183} C_DIS
LIN {X -3.8698,Y -134.7081,Z 161,A -93.5457,B 20.6493,C -0.5398,E1 20.651,E2 541.5716} C_DIS
LIN {X -7.3438,Y -134.5646,Z 161,A -94.9833,B 20.6493,C -0.5415,E1 20.647,E2 543.0048} C_DIS
LIN {X -10.5761,Y -134.3501,Z 161,A -96.3633,B 20.6493,C -0.5415,E1 20.6431,E2 544.3858} C_DIS
LIN {X -13.4635,Y -134.0906,Z 161,A -97.5829,B 20.6493,C -0.5421,E1 20.6397,E2 545.6041} C_DIS
LIN {X -16.1284,Y -133.795,Z 161,A -98.7394,B 20.6493,C -0.5416,E1 20.6365,E2 546.763} C_DIS
LIN {X -19.4889,Y -133.3475,Z 161,A -100.2109,B 20.6493,C -0.5406,E1 20.6324,E2 548.2386} C_DIS
LIN {X -22.7728,Y -132.8267,Z 161,A -101.6027,B 20.6493,C -0.542,E1 20.6286,E2 549.6282} C_DIS
LIN {X -25.9007,Y -132.2524,Z 161,A -102.9443,B 20.6493,C -0.543,E1 20.6249,E2 550.9687} C_DIS
LIN {X -28.7625,Y -131.6586,Z 161,A -104.2316,B 20.6493,C -0.5417,E1 20.6214,E2 552.2617} C_DIS
LIN {X -32.1782,Y -130.8667,Z 161,A -105.7076,B 20.6493,C -0.5431,E1 20.6174,E2 553.736} C_DIS
LIN {X -34.8992,Y -130.1661,Z 161,A -106.92,B 20.6493,C -0.5431,E1 20.6141,E2 554.9507} C_DIS
LIN {X -38.3661,Y -129.1876,Z 161,A -108.4219,B 20.6493,C -0.5454,E1 20.6101,E2 556.4491} C_DIS
LIN {X -41.7931,Y -128.1216,Z 161,A -109.9652,B 20.6493,C -0.5458,E1 20.606,E2 557.9945} C_DIS
LIN {X -44.7391,Y -127.1217,Z 161,A -111.3005,B 20.6493,C -0.5464,E1 20.6024,E2 559.3313} C_DIS
LIN {X -47.7102,Y -126.0359,Z 161,A -112.6318,B 20.6492,C -0.5483,E1 20.599,E2 560.6607} C_DIS
LIN {X -50.9742,Y -124.7523,Z 161,A -114.139,B 20.6492,C -0.5491,E1 20.5951,E2 562.1697} C_DIS
LIN {X -54.0694,Y -123.4423,Z 161,A -115.5575,B 20.6492,C -0.5511,E1 20.5914,E2 563.5867} C_DIS
LIN {X -57.3288,Y -121.964,Z 161,A -117.1006,B 20.6491,C -0.5519,E1 20.5875,E2 565.1322} C_DIS
LIN {X -59.9532,Y -120.6931,Z 161,A -118.3854,B 20.6491,C -0.5515,E1 20.5843,E2 566.4221} C_DIS
LIN {X -63.4067,Y -118.9176,Z 161,A -119.9929,B 20.6491,C -0.5555,E1 20.5803,E2 568.0239} C_DIS
LIN {X -66.579,Y -117.1704,Z 161,A -121.6636,B 20.6491,C -0.5521,E1 20.5762,E2 569.7102} C_DIS
LIN {X -70.1029,Y -115.0973,Z 161,A -123.3993,B 20.6491,C -0.5548,E1 20.572,E2 571.4449} C_DIS
LIN {X -73.7451,Y -112.7983,Z 161,A -125.2296,B 20.6489,C -0.5576,E1 20.5677,E2 573.2743} C_DIS
LIN {X -77.2388,Y -110.435,Z 161,A -127.0118,B 20.6489,C -0.561,E1 20.5636,E2 575.0542} C_DIS
LIN {X -80.8326,Y -107.8327,Z 161,A -128.9349,B 20.6489,C -0.5628,E1 20.5593,E2 576.9808} C_DIS
LIN {X -84.2656,Y -105.1718,Z 161,A -130.6881,B 20.6486,C -0.57,E1 20.5555,E2 578.7214} C_DIS
LIN {X -87.0328,Y -102.8932,Z 161,A -132.3461,B 20.6486,C -0.5673,E1 20.5519,E2 580.3949} C_DIS
LIN {X -90.3126,Y -100.0268,Z 161,A -134.2077,B 20.6486,C -0.5706,E1 20.548,E2 582.2564} C_DIS
LIN {X -93.5689,Y -96.9873,Z 161,A -136.089,B 20.6485,C -0.575,E1 20.5442,E2 584.1347} C_DIS
LIN {X -96.4079,Y -94.1658,Z 161,A -137.743,B 20.6483,C -0.5805,E1 20.541,E2 585.7816} C_DIS
LIN {X -99.3708,Y -91.0336,Z 161,A -139.5932,B 20.6483,C -0.5838,E1 20.5375,E2 587.6324} C_DIS
LIN {X -102.3287,Y -87.6958,Z 161,A -141.4298,B 20.6481,C -0.5906,E1 20.5341,E2 589.4601} C_DIS
LIN {X -104.6911,Y -84.8617,Z 161,A -143.1496,B 20.6481,C -0.5881,E1 20.531,E2 591.1969} C_DIS
LIN {X -107.2468,Y -81.6079,Z 161,A -144.8322,B 20.6479,C -0.5954,E1 20.5282,E2 592.8684} C_DIS
LIN {X -109.8166,Y -78.1155,Z 161,A -146.6586,B 20.6478,C -0.6006,E1 20.5252,E2 594.6909} C_DIS
LIN {X -112.1611,Y -74.7096,Z 161,A -148.4552,B 20.6478,C -0.6035,E1 20.5224,E2 596.4904} C_DIS
LIN {X -114.4754,Y -71.1127,Z 161,A -150.3175,B 20.6476,C -0.6064,E1 20.5196,E2 598.3561} C_DIS
LIN {X -116.7948,Y -67.2362,Z 161,A -152.1882,B 20.6474,C -0.6135,E1 20.5169,E2 600.2185} C_DIS
LIN {X -118.5135,Y -64.1587,Z 161,A -153.807,B 20.6474,C -0.6127,E1 20.5147,E2 601.8503} C_DIS
LIN {X -120.39,Y -60.562,Z 161,A -155.403,B 20.6472,C -0.6226,E1 20.5127,E2 603.4285} C_DIS
LIN {X -121.8767,Y -57.5115,Z 161,A -156.8711,B 20.6471,C -0.6256,E1 20.5109,E2 604.8979} C_DIS
LIN {X -123.3625,Y -54.2541,Z 161,A -158.4029,B 20.647,C -0.6294,E1 20.5092,E2 606.429} C_DIS
LIN {X -124.536,Y -51.4986,Z 161,A -159.6749,B 20.6469,C -0.6332,E1 20.5078,E2 607.6992} C_DIS
LIN {X -125.9089,Y -48.0495,Z 161,A -161.272,B 20.6468,C -0.6369,E1 20.5062,E2 609.2966} C_DIS
LIN {X -126.8727,Y -45.4369,Z 161,A -162.4684,B 20.6467,C -0.6399,E1 20.5051,E2 610.4929} C_DIS
LIN {X -128.0592,Y -41.9805,Z 161,A -164.0268,B 20.6465,C -0.6443,E1 20.5037,E2 612.0498} C_DIS
LIN {X -129.1035,Y -38.6533,Z 161,A -165.5188,B 20.6465,C -0.6483,E1 20.5024,E2 613.541} C_DIS
LIN {X -129.9507,Y -35.6978,Z 161,A -166.8337,B 20.6463,C -0.6519,E1 20.5015,E2 614.855} C_DIS
LIN {X -130.7467,Y -32.6605,Z 161,A -168.1955,B 20.6463,C -0.6549,E1 20.5005,E2 616.2181} C_DIS
LIN {X -131.5589,Y -29.2243,Z 161,A -169.6876,B 20.6461,C -0.6598,E1 20.4996,E2 617.707} C_DIS
LIN {X -132.1785,Y -26.2752,Z 161,A -170.9846,B 20.646,C -0.6632,E1 20.4989,E2 619.0039} C_DIS
LIN {X -132.7956,Y -22.9593,Z 161,A -172.4199,B 20.6458,C -0.6675,E1 20.4981,E2 620.4374} C_DIS
LIN {X -133.5192,Y -18.2871,Z 161,A -174.4428,B 20.6457,C -0.6733,E1 20.4973,E2 622.4588} C_DIS
LIN {X -133.8849,Y -15.3746,Z 161,A -175.6982,B 20.6455,C -0.6769,E1 20.4969,E2 623.7132} C_DIS
LIN {X -134.2206,Y -12.1093,Z 161,A -177.2359,B 20.6455,C -0.6756,E1 20.4965,E2 625.2659} C_DIS
LIN {X -134.5069,Y -8.3139,Z 161,A -178.7704,B 20.6453,C -0.684,E1 20.4962,E2 626.7877} C_DIS
LIN {X -134.6805,Y -4.7575,Z 161,A 179.7418,B 20.6451,C -0.6898,E1 20.496,E2 628.2701} C_DIS
LIN {X -134.7575,Y -1.4923,Z 161,A 178.3867,B 20.6449,C -0.6956,E1 20.496,E2 629.6189} C_DIS
LIN {X -134.7592,Y 1.2375,Z 161,A 177.0133,B 20.6451,C -0.6908,E1 20.496,E2 631.0161} C_DIS
LIN {X -134.6621,Y 5.2295,Z 161,A 175.4299,B 20.6448,C -0.7007,E1 20.496,E2 632.583} C_DIS
LIN {X -134.4864,Y 8.6457,Z 161,A 173.9616,B 20.6446,C -0.7048,E1 20.4963,E2 634.0506} C_DIS
LIN {X -134.236,Y 11.9261,Z 161,A 172.5816,B 20.6445,C -0.71,E1 20.4966,E2 635.4262} C_DIS
LIN {X -133.9069,Y 15.1898,Z 161,A 171.1729,B 20.6443,C -0.7138,E1 20.4971,E2 636.8344} C_DIS
LIN {X -133.3716,Y 19.3199,Z 161,A 169.334,B 20.6443,C -0.7167,E1 20.4978,E2 638.6785} C_DIS
LIN {X -132.8267,Y 22.7728,Z 161,A 167.8844,B 20.644,C -0.7229,E1 20.4984,E2 640.1213} C_DIS
LIN {X -132.3148,Y 25.5743,Z 161,A 166.6119,B 20.644,C -0.7242,E1 20.4991,E2 641.3991} C_DIS
LIN {X -131.5589,Y 29.2243,Z 161,A 165.062,B 20.6438,C -0.7306,E1 20.5,E2 642.9423} C_DIS
LIN {X -130.8667,Y 32.1782,Z 161,A 163.7794,B 20.6436,C -0.7349,E1 20.5008,E2 644.2219} C_DIS
LIN {X -130.0032,Y 35.5099,Z 161,A 162.2826,B 20.6436,C -0.7381,E1 20.5019,E2 645.7203} C_DIS
LIN {X -129.1585,Y 38.4655,Z 161,A 160.9634,B 20.6434,C -0.7417,E1 20.5029,E2 647.0388} C_DIS
LIN {X -128.1216,Y 41.7931,Z 161,A 159.4681,B 20.6433,C -0.7457,E1 20.5042,E2 648.5332} C_DIS
LIN {X -127.1345,Y 44.7021,Z 161,A 158.1388,B 20.6432,C -0.7487,E1 20.5054,E2 649.8631} C_DIS
LIN {X -125.9787,Y 47.8631,Z 161,A 156.7065,B 20.643,C -0.753,E1 20.5068,E2 651.2933} C_DIS
LIN {X -124.7523,Y 50.9742,Z 161,A 155.272,B 20.6429,C -0.7568,E1 20.5083,E2 652.7269} C_DIS
LIN {X -123.5416,Y 53.8396,Z 161,A 153.9423,B 20.6428,C -0.7604,E1 20.5097,E2 654.0553} C_DIS
LIN {X -121.964,Y 57.3288,Z 161,A 152.2964,B 20.6426,C -0.7645,E1 20.5117,E2 655.7007} C_DIS
LIN {X -120.572,Y 60.1987,Z 161,A 150.9205,B 20.6425,C -0.7677,E1 20.5134,E2 657.0767} C_DIS
LIN {X -118.5618,Y 64.0688,Z 161,A 149.048,B 20.6423,C -0.7723,E1 20.5158,E2 658.9484} C_DIS
LIN {X -116.7948,Y 67.2362,Z 161,A 147.3802,B 20.6423,C -0.7716,E1 20.5181,E2 660.6288} C_DIS
LIN {X -114.4612,Y 71.1355,Z 161,A 145.4762,B 20.6421,C -0.7781,E1 20.5209,E2 662.5263} C_DIS
LIN {X -112.3236,Y 74.4661,Z 161,A 143.755,B 20.6421,C -0.7812,E1 20.5235,E2 664.2495} C_DIS
LIN {X -109.9491,Y 77.9288,Z 161,A 141.9894,B 20.6418,C -0.7868,E1 20.5263,E2 666.0099} C_DIS
LIN {X -107.3723,Y 81.4426,Z 161,A 140.1588,B 20.6416,C -0.7926,E1 20.5293,E2 667.835} C_DIS
LIN {X -104.6911,Y 84.8617,Z 161,A 138.3383,B 20.6414,C -0.7984,E1 20.5325,E2 669.6495} C_DIS
LIN {X -102.3966,Y 87.6169,Z 161,A 136.692,B 20.6414,C -0.7973,E1 20.5355,E2 671.3081} C_DIS
LIN {X -99.4405,Y 90.9577,Z 161,A 134.7683,B 20.6413,C -0.8009,E1 20.5391,E2 673.2321} C_DIS
LIN {X -96.5917,Y 93.9774,Z 161,A 133.1191,B 20.641,C -0.8098,E1 20.5422,E2 674.8648} C_DIS
LIN {X -94.1267,Y 96.4462,Z 161,A 131.6154,B 20.6409,C -0.8125,E1 20.5452,E2 676.3688} C_DIS
LIN {X -91.1456,Y 99.2678,Z 161,A 129.7924,B 20.6409,C -0.8133,E1 20.549,E2 678.1986} C_DIS
LIN {X -87.6958,Y 102.3287,Z 161,A 127.8886,B 20.6406,C -0.8199,E1 20.5529,E2 680.0927} C_DIS
LIN {X -84.8617,Y 104.6911,Z 161,A 126.1974,B 20.6406,C -0.8183,E1 20.5566,E2 681.7966} C_DIS
LIN {X -81.6079,Y 107.2468,Z 161,A 124.5558,B 20.6403,C -0.8267,E1 20.5602,E2 683.4216} C_DIS
LIN {X -78.736,Y 109.3729,Z 161,A 123.0296,B 20.6403,C -0.8294,E1 20.5636,E2 684.9467} C_DIS
LIN {X -75.9003,Y 111.3595,Z 161,A 121.5511,B 20.6401,C -0.832,E1 20.567,E2 686.4241} C_DIS
LIN {X -72.509,Y 113.5962,Z 161,A 119.7957,B 20.6401,C -0.8341,E1 20.5712,E2 688.1806} C_DIS
LIN {X -69.2792,Y 115.5946,Z 161,A 118.0714,B 20.6401,C -0.8325,E1 20.5753,E2 689.9161} C_DIS
LIN {X -65.6571,Y 117.69,Z 161,A 116.3828,B 20.6398,C -0.8392,E1 20.5794,E2 691.5916} C_DIS
LIN {X -62.0776,Y 119.6155,Z 161,A 114.6754,B 20.6397,C -0.8429,E1 20.5836,E2 693.2944} C_DIS
LIN {X -58.8578,Y 121.2335,Z 161,A 113.1398,B 20.6397,C -0.8451,E1 20.5874,E2 694.8288} C_DIS
LIN {X -56.1909,Y 122.4901,Z 161,A 111.8489,B 20.6396,C -0.8454,E1 20.5907,E2 696.1228} C_DIS
LIN {X -52.7092,Y 124.0304,Z 161,A 110.2603,B 20.6395,C -0.8489,E1 20.5947,E2 697.706} C_DIS
LIN {X -49.6065,Y 125.3036,Z 161,A 108.8311,B 20.6394,C -0.8506,E1 20.5984,E2 699.1342} C_DIS
LIN {X -46.5995,Y 126.452,Z 161,A 107.4622,B 20.6394,C -0.8523,E1 20.602,E2 700.5017} C_DIS
LIN {X -43.3607,Y 127.5996,Z 161,A 105.9965,B 20.6393,C -0.8539,E1 20.6059,E2 701.9665} C_DIS
LIN {X -40.4114,Y 128.5629,Z 161,A 104.6676,B 20.6393,C -0.8549,E1 20.6094,E2 703.2954} C_DIS
LIN {X -37.0819,Y 129.5636,Z 161,A 103.1954,B 20.6391,C -0.8567,E1 20.6133,E2 704.7655} C_DIS
LIN {X -34.451,Y 130.2856,Z 161,A 102.0329,B 20.6391,C -0.8578,E1 20.6165,E2 705.9272} C_DIS
LIN {X -31.2184,Y 131.098,Z 161,A 100.581,B 20.6391,C -0.8576,E1 20.6204,E2 707.3822} C_DIS
LIN {X -27.8428,Y 131.8571,Z 161,A 99.1444,B 20.6391,C -0.8602,E1 20.6243,E2 708.8134} C_DIS
LIN {X -24.5224,Y 132.5159,Z 161,A 97.7043,B 20.639,C -0.8612,E1 20.6283,E2 710.2526} C_DIS
LIN {X -20.4727,Y 133.1994,Z 161,A 95.9442,B 20.639,C -0.8618,E1 20.6331,E2 712.0129} C_DIS
LIN {X -16.7365,Y 133.7224,Z 161,A 94.3552,B 20.6389,C -0.8633,E1 20.6375,E2 713.5991} C_DIS
LIN {X -14.2829,Y 134.0045,Z 161,A 93.2565,B 20.6389,C -0.8618,E1 20.6406,E2 714.7029} C_DIS
LIN {X -10.9911,Y 134.315,Z 161,A 91.9195,B 20.6389,C -0.8654,E1 20.6443,E2 716.0307} C_DIS
LIN {X -7.5251,Y 134.5555,Z 161,A 90.4248,B 20.6389,C -0.8651,E1 20.6484,E2 717.5267} C_DIS
LIN {X -4.6772,Y 134.6836,Z 161,A 89.2148,B 20.6388,C -0.8655,E1 20.6518,E2 718.7358} C_DIS
LIN {X -1.4923,Y 134.7575,Z 161,A 87.8618,B 20.6388,C -0.8659,E1 20.6556,E2 720.0879} C_DIS
LIN {X 2.1371,Y 134.7467,Z 161,A 86.2649,B 20.6388,C -0.8638,E1 20.6601,E2 721.6905} C_DIS
LIN {X 6.0079,Y 134.6317,Z 161,A 84.6668,B 20.6388,C -0.8659,E1 20.6645,E2 723.2822} C_DIS
LIN {X 8.8659,Y 134.4729,Z 161,A 83.4397,B 20.6388,C -0.8654,E1 20.6679,E2 724.51} C_DIS
LIN {X 11.7436,Y 134.2515,Z 161,A 82.2362,B 20.6388,C -0.8663,E1 20.6713,E2 725.7102} C_DIS
LIN {X 14.7573,Y 133.9535,Z 161,A 80.9126,B 20.6388,C -0.8645,E1 20.675,E2 727.0377} C_DIS
LIN {X 18.1018,Y 133.5435,Z 161,A 79.4945,B 20.6388,C -0.8648,E1 20.6789,E2 728.4537} C_DIS
LIN {X 21.3988,Y 133.056,Z 161,A 78.0767,B 20.6388,C -0.8643,E1 20.6828,E2 729.8713} C_DIS
LIN {X 24.2965,Y 132.5563,Z 161,A 76.8299,B 20.6388,C -0.8639,E1 20.6862,E2 731.1174} C_DIS
LIN {X 27.6552,Y 131.8976,Z 161,A 75.3697,B 20.6388,C -0.863,E1 20.6902,E2 732.578} C_DIS
LIN {X 30.607,Y 131.243,Z 161,A 74.0874,B 20.6389,C -0.8624,E1 20.6937,E2 733.8597} C_DIS
LIN {X 33.4365,Y 130.5497,Z 161,A 72.8326,B 20.6389,C -0.861,E1 20.6971,E2 735.1163} C_DIS
LIN {X 36.8118,Y 129.6391,Z 161,A 71.3544,B 20.639,C -0.8603,E1 20.7011,E2 736.5934} C_DIS
LIN {X 40.0362,Y 128.6803,Z 161,A 69.9226,B 20.639,C -0.8591,E1 20.7049,E2 738.0255} C_DIS
LIN {X 43.0101,Y 127.7163,Z 161,A 68.6236,B 20.639,C -0.8593,E1 20.7083,E2 739.3208} C_DIS
LIN {X 46.079,Y 126.6412,Z 161,A 67.2003,B 20.6392,C -0.8562,E1 20.7121,E2 740.7491} C_DIS
LIN {X 49.4205,Y 125.3759,Z 161,A 65.7043,B 20.6392,C -0.8557,E1 20.716,E2 742.2426} C_DIS
LIN {X 52.244,Y 124.2247,Z 161,A 64.3805,B 20.6392,C -0.8532,E1 20.7194,E2 743.5699} C_DIS
LIN {X 55.4857,Y 122.8116,Z 161,A 62.9191,B 20.6392,C -0.8532,E1 20.7231,E2 745.0264} C_DIS
LIN {X 58.8578,Y 121.2335,Z 161,A 61.3298,B 20.6394,C -0.851,E1 20.7271,E2 746.6169} C_DIS
LIN {X 61.8972,Y 119.7102,Z 161,A 59.8302,B 20.6395,C -0.8468,E1 20.7309,E2 748.1236} C_DIS
LIN {X 65.6571,Y 117.69,Z 161,A 58.0506,B 20.6395,C -0.8458,E1 20.7352,E2 749.8995} C_DIS
LIN {X 69.2792,Y 115.5946,Z 161,A 56.2926,B 20.6396,C -0.8441,E1 20.7395,E2 751.6556} C_DIS
LIN {X 72.3823,Y 113.6773,Z 161,A 54.6342,B 20.6399,C -0.8369,E1 20.7434,E2 753.3278} C_DIS
LIN {X 75.9999,Y 111.2912,Z 161,A 52.8021,B 20.64,C -0.8344,E1 20.7477,E2 755.1595} C_DIS
LIN {X 79.4378,Y 108.8643,Z 161,A 51.0233,B 20.6401,C -0.8317,E1 20.7517,E2 756.938} C_DIS
LIN {X 82.9836,Y 106.1859,Z 161,A 49.1337,B 20.6403,C -0.8283,E1 20.7559,E2 758.8287} C_DIS
LIN {X 86.2064,Y 103.5865,Z 161,A 47.4667,B 20.6403,C -0.8292,E1 20.7595,E2 760.4855} C_DIS
LIN {X 89.5082,Y 100.7473,Z 161,A 45.6239,B 20.6403,C -0.8259,E1 20.7634,E2 762.3284} C_DIS
LIN {X 92.7194,Y 97.7999,Z 161,A 43.8192,B 20.6404,C -0.8243,E1 20.767,E2 764.1285} C_DIS
LIN {X 95.5438,Y 95.0421,Z 161,A 42.0676,B 20.6407,C -0.8175,E1 20.7705,E2 765.8904} C_DIS
LIN {X 98.5478,Y 91.9236,Z 161,A 40.2306,B 20.6408,C -0.8136,E1 20.7741,E2 767.7283} C_DIS
LIN {X 101.6201,Y 88.5155,Z 161,A 38.3089,B 20.6409,C -0.8105,E1 20.7776,E2 769.6482} C_DIS
LIN {X 104.56,Y 85.0231,Z 161,A 36.4392,B 20.6409,C -0.8092,E1 20.7809,E2 771.5109} C_DIS
LIN {X 107.0999,Y 81.8,Z 161,A 34.6414,B 20.6412,C -0.8026,E1 20.784,E2 773.3169} C_DIS
LIN {X 109.8166,Y 78.1155,Z 161,A 32.6917,B 20.6414,C -0.7976,E1 20.7872,E2 775.269} C_DIS
LIN {X 112.3236,Y 74.4661,Z 161,A 30.8897,B 20.6414,C -0.7965,E1 20.79,E2 777.0631} C_DIS
LIN {X 114.5931,Y 70.9235,Z 161,A 29.0997,B 20.6416,C -0.7918,E1 20.7927,E2 778.8552} C_DIS
LIN {X 116.7948,Y 67.2362,Z 161,A 27.3145,B 20.6417,C -0.7888,E1 20.7952,E2 780.6374} C_DIS
LIN {X 118.5618,Y 64.0688,Z 161,A 25.6735,B 20.6421,C -0.7801,E1 20.7975,E2 782.2923} C_DIS
LIN {X 120.39,Y 60.562,Z 161,A 24.1189,B 20.6421,C -0.7813,E1 20.7994,E2 783.8333} C_DIS
LIN {X 121.8767,Y 57.5115,Z 161,A 22.7131,B 20.6421,C -0.779,E1 20.8011,E2 785.2363} C_DIS
LIN {X 123.2726,Y 54.455,Z 161,A 21.2692,B 20.6423,C -0.7743,E1 20.8028,E2 786.6839} C_DIS
LIN {X 124.6774,Y 51.1599,Z 161,A 19.7682,B 20.6423,C -0.7709,E1 20.8044,E2 788.1841} C_DIS
LIN {X 125.7176,Y 48.5414,Z 161,A 18.5707,B 20.6425,C -0.7675,E1 20.8056,E2 789.3831} C_DIS
LIN {X 126.9895,Y 45.113,Z 161,A 17.049,B 20.6426,C -0.7645,E1 20.8071,E2 790.9028} C_DIS
LIN {X 128.0592,Y 41.9805,Z 161,A 15.6439,B 20.6428,C -0.7604,E1 20.8083,E2 792.3096} C_DIS
LIN {X 129.1035,Y 38.6533,Z 161,A 14.1742,B 20.6428,C -0.7566,E1 20.8095,E2 793.7798} C_DIS
LIN {X 129.9068,Y 35.8548,Z 161,A 12.9463,B 20.643,C -0.7533,E1 20.8105,E2 795.0081} C_DIS
LIN {X 130.7737,Y 32.5538,Z 161,A 11.5018,B 20.6431,C -0.7492,E1 20.8115,E2 796.4539} C_DIS
LIN {X 131.5589,Y 29.2243,Z 161,A 10.0688,B 20.6433,C -0.7457,E1 20.8123,E2 797.8864} C_DIS
LIN {X 132.1502,Y 26.4141,Z 161,A 8.8601,B 20.6433,C -0.7426,E1 20.813,E2 799.0952} C_DIS
LIN {X 132.7114,Y 23.4295,Z 161,A 7.5973,B 20.6435,C -0.7399,E1 20.8137,E2 800.3564} C_DIS
LIN {X 133.2683,Y 20.0274,Z 161,A 6.1208,B 20.6436,C -0.7348,E1 20.8143,E2 801.8365} C_DIS
LIN {X 133.711,Y 16.8234,Z 161,A 4.7705,B 20.6437,C -0.7317,E1 20.8148,E2 803.1859} C_DIS
LIN {X 134.021,Y 14.1301,Z 161,A 3.5814,B 20.6439,C -0.7264,E1 20.8152,E2 804.3812} C_DIS
LIN {X 134.3501,Y 10.5761,Z 161,A 2.1219,B 20.6439,C -0.7243,E1 20.8155,E2 805.8359} C_DIS
LIN {X 134.5555,Y 7.5251,Z 161,A 0.8343,B 20.6441,C -0.7208,E1 20.8157,E2 807.124} C_DIS
LIN {X 134.6907,Y 4.4965,Z 161,A -0.6073,B 20.6445,C -0.7095,E1 20.8159,E2 808.5866} C_DIS
LIN {X 134.7632,Y 0.5677,Z 161,A -2.1443,B 20.6445,C -0.7105,E1 20.8159,E2 810.1096} C_DIS
LIN {X 134.7325,Y -2.9913,Z 161,A -3.6004,B 20.6445,C -0.7083,E1 20.8159,E2 811.5611} C_DIS
LIN {X 134.6317,Y -6.0079,Z 161,A -4.8757,B 20.6446,C -0.7046,E1 20.8157,E2 812.8375} C_DIS
LIN {X 134.3681,Y -10.3297,Z 161,A -6.6862,B 20.6448,C -0.7002,E1 20.8154,E2 814.6472} C_DIS
LIN {X 134.0906,Y -13.4635,Z 161,A -8.0424,B 20.645,C -0.6951,E1 20.8151,E2 816.0078} C_DIS
LIN {X 133.7224,Y -16.7365,Z 161,A -9.4263,B 20.645,C -0.6914,E1 20.8146,E2 817.392} C_DIS
LIN {X 133.3237,Y -19.6555,Z 161,A -10.6792,B 20.6452,C -0.6874,E1 20.8141,E2 818.647} C_DIS
LIN {X 132.8267,Y -22.7728,Z 161,A -12.0052,B 20.6453,C -0.6839,E1 20.8135,E2 819.9732} C_DIS
LIN {X 132.2524,Y -25.9007,Z 161,A -13.3567,B 20.6454,C -0.6797,E1 20.8128,E2 821.3269} C_DIS
LIN {X 131.3273,Y -30.238,Z 161,A -15.2634,B 20.6457,C -0.6728,E1 20.8117,E2 823.2394} C_DIS
LIN {X 130.4967,Y -33.6452,Z 161,A -16.7013,B 20.6457,C -0.6706,E1 20.8107,E2 824.6731} C_DIS
LIN {X 129.5636,Y -37.0819,Z 161,A -18.2081,B 20.6459,C -0.6662,E1 20.8096,E2 826.1817} C_DIS
LIN {X 128.6803,Y -40.0362,Z 161,A -19.5125,B 20.6459,C -0.6625,E1 20.8085,E2 827.4874} C_DIS
LIN {X 127.7873,Y -42.7969,Z 161,A -20.7451,B 20.6461,C -0.6587,E1 20.8074,E2 828.7218} C_DIS
LIN {X 126.5617,Y -46.2994,Z 161,A -22.3046,B 20.6462,C -0.6547,E1 20.8059,E2 830.2818} C_DIS
LIN {X 125.3759,Y -49.4205,Z 161,A -23.7147,B 20.6463,C -0.6509,E1 20.8045,E2 831.6931} C_DIS
LIN {X 124.1077,Y -52.524,Z 161,A -25.131,B 20.6465,C -0.647,E1 20.803,E2 833.1106} C_DIS
LIN {X 122.756,Y -55.61,Z 161,A -26.5623,B 20.6465,C -0.6428,E1 20.8014,E2 834.5442} C_DIS
LIN {X 121.2335,Y -58.8578,Z 161,A -28.0691,B 20.6467,C -0.6391,E1 20.7996,E2 836.0513} C_DIS
LIN {X 119.7102,Y -61.8972,Z 161,A -29.5054,B 20.6467,C -0.6354,E1 20.7977,E2 837.4888} C_DIS
LIN {X 118.1533,Y -64.8192,Z 161,A -30.9041,B 20.6469,C -0.6317,E1 20.7959,E2 838.8886} C_DIS
LIN {X 116.3645,Y -67.978,Z 161,A -32.5605,B 20.6472,C -0.6221,E1 20.7936,E2 840.5616} C_DIS
LIN {X 114.1377,Y -71.6541,Z 161,A -34.3767,B 20.6473,C -0.6175,E1 20.7909,E2 842.3795} C_DIS
LIN {X 111.9013,Y -75.0987,Z 161,A -35.9884,B 20.6473,C -0.6189,E1 20.7884,E2 843.9773} C_DIS
LIN {X 109.9365,Y -77.9467,Z 161,A -37.4494,B 20.6473,C -0.6154,E1 20.7861,E2 845.4394} C_DIS
LIN {X 107.675,Y -81.0416,Z 161,A -39.1709,B 20.6476,C -0.6068,E1 20.7832,E2 847.1749} C_DIS
LIN {X 105.1718,Y -84.2656,Z 161,A -40.7942,B 20.6476,C -0.6074,E1 20.7804,E2 848.7869} C_DIS
LIN {X 102.9606,Y -86.9535,Z 161,A -42.3592,B 20.6478,C -0.5997,E1 20.7776,E2 850.3648} C_DIS
LIN {X 100.1147,Y -90.2154,Z 161,A -44.1453,B 20.6478,C -0.5976,E1 20.7743,E2 852.147} C_DIS
LIN {X 97.1979,Y -93.3504,Z 161,A -45.9152,B 20.6479,C -0.5955,E1 20.7709,E2 853.9133} C_DIS
LIN {X 94.675,Y -95.9085,Z 161,A -47.4223,B 20.648,C -0.5928,E1 20.7679,E2 855.4201} C_DIS
LIN {X 92.1609,Y -98.3268,Z 161,A -49.0055,B 20.6482,C -0.5847,E1 20.7647,E2 857.018} C_DIS
LIN {X 88.8549,Y -101.3239,Z 161,A -50.9074,B 20.6484,C -0.5802,E1 20.7607,E2 858.9231} C_DIS
LIN {X 85.6163,Y -104.0752,Z 161,A -52.5793,B 20.6483,C -0.5824,E1 20.7572,E2 860.5808} C_DIS
LIN {X 82.9019,Y -106.2501,Z 161,A -54.1567,B 20.6485,C -0.5748,E1 20.7537,E2 862.1725} C_DIS
LIN {X 79.4441,Y -108.8597,Z 161,A -55.9624,B 20.6485,C -0.5727,E1 20.7497,E2 863.9762} C_DIS
LIN {X 75.9003,Y -111.3595,Z 161,A -57.7423,B 20.6485,C -0.5719,E1 20.7456,E2 865.7507} C_DIS
LIN {X 72.3823,Y -113.6773,Z 161,A -59.4967,B 20.6486,C -0.5702,E1 20.7415,E2 867.5027} C_DIS
LIN {X 69.2792,Y -115.5946,Z 161,A -61.1621,B 20.6488,C -0.5622,E1 20.7375,E2 869.1843} C_DIS
LIN {X 65.6571,Y -117.69,Z 161,A -62.8363,B 20.6488,C -0.5639,E1 20.7334,E2 870.8477} C_DIS
LIN {X 62.0776,Y -119.6155,Z 161,A -64.5285,B 20.6488,C -0.5626,E1 20.7293,E2 872.5374} C_DIS
LIN {X 58.8578,Y -121.2335,Z 161,A -66.0532,B 20.6488,C -0.5605,E1 20.7254,E2 874.063} C_DIS
LIN {X 56.1214,Y -122.5223,Z 161,A -67.3568,B 20.6489,C -0.5578,E1 20.7221,E2 875.3702} C_DIS
LIN {X 52.7092,Y -124.0304,Z 161,A -68.9116,B 20.6489,C -0.5569,E1 20.7182,E2 876.9229} C_DIS
LIN {X 49.6065,Y -125.3036,Z 161,A -70.3311,B 20.649,C -0.5552,E1 20.7145,E2 878.3432} C_DIS
LIN {X 46.4893,Y -126.4933,Z 161,A -71.7433,B 20.649,C -0.5537,E1 20.7108,E2 879.756} C_DIS
LIN {X 43.5593,Y -127.5307,Z 161,A -73.0594,B 20.649,C -0.5523,E1 20.7073,E2 881.0728} C_DIS
LIN {X 40.4114,Y -128.5629,Z 161,A -74.4693,B 20.6491,C -0.5506,E1 20.7036,E2 882.4841} C_DIS
LIN {X 37.3317,Y -129.4905,Z 161,A -75.8269,B 20.6491,C -0.5496,E1 20.6999,E2 883.8418} C_DIS
LIN {X 34.1257,Y -130.3724,Z 161,A -77.205,B 20.6491,C -0.5497,E1 20.6962,E2 885.2167} C_DIS
LIN {X 31.2819,Y -131.0827,Z 161,A -78.4916,B 20.6492,C -0.5467,E1 20.6927,E2 886.5094} C_DIS
LIN {X 28.2083,Y -131.7782,Z 161,A -79.8475,B 20.6492,C -0.5449,E1 20.689,E2 887.8685} C_DIS
LIN {X 24.5224,Y -132.5159,Z 161,A -81.4004,B 20.6492,C -0.5456,E1 20.6848,E2 889.4171} C_DIS
LIN {X 21.9437,Y -132.965,Z 161,A -82.5477,B 20.6493,C -0.5433,E1 20.6816,E2 890.5694} C_DIS
LIN {X 18.2871,Y -133.5192,Z 161,A -84.0766,B 20.6493,C -0.5441,E1 20.6774,E2 892.0941} C_DIS
LIN {X 15.7752,Y -133.8371,Z 161,A -85.1947,B 20.6493,C -0.5417,E1 20.6742,E2 893.2181} C_DIS
LIN {X 12.1093,Y -134.2206,Z 161,A -86.7114,B 20.6493,C -0.5431,E1 20.67,E2 894.7297} C_DIS
LIN {X 9.4153,Y -134.4348,Z 161,A -87.8577,B 20.6493,C -0.5427,E1 20.6669,E2 895.8762} C_DIS
LIN {X 6.0079,Y -134.6317,Z 161,A -89.3042,B 20.6493,C -0.5424,E1 20.6628,E2 897.323} C_DIS
LIN {X 3.1712,Y -134.7275,Z 161,A -90.5146,B 20.6493,C -0.5419,E1 20.6594,E2 898.5346} C_DIS
LIN {X 3.1712,Y -134.7275,Z 161,A -90.5146,B 20.6493,C -0.5419,E1 20.6594,E2 898.5346} C_DIS
Enddeposition()
LIN {X 0.9612,Y -133.8342,Z 161,A -90.5315,B 19.4805,C -0.4202,E1 19.4874,E2 898.8002} C_DIS
Startdeposition()
$VEL.CP = VEL_PRINT
LIN {X 4.2906,Y -133.7718,Z 161,A -89.1185,B 19.4805,C -0.42,E1 19.4914,E2 897.3882} C_DIS
LIN {X 7.1731,Y -133.6478,Z 161,A -87.7058,B 19.4804,C -0.4278,E1 19.4954,E2 895.9526} C_DIS
LIN {X 11.3121,Y -133.3604,Z 161,A -85.9589,B 19.4804,C -0.4274,E1 19.5002,E2 894.2082} C_DIS
LIN {X 15.8341,Y -132.8993,Z 161,A -84.0843,B 19.4804,C -0.4254,E1 19.5054,E2 892.3412} C_DIS
LIN {X 18.9753,Y -132.4873,Z 161,A -82.7687,B 19.4804,C -0.4246,E1 19.509,E2 891.0297} C_DIS
LIN {X 22.3168,Y -131.9658,Z 161,A -81.3295,B 19.4804,C -0.4252,E1 19.513,E2 889.5905} C_DIS
LIN {X 25.8718,Y -131.3169,Z 161,A -79.7951,B 19.4804,C -0.4258,E1 19.5172,E2 888.0566} C_DIS
LIN {X 28.4844,Y -130.7731,Z 161,A -78.6645,B 19.4804,C -0.4263,E1 19.5203,E2 886.9264} C_DIS
LIN {X 31.5936,Y -130.0569,Z 161,A -77.2639,B 19.4804,C -0.429,E1 19.5241,E2 885.5203} C_DIS
LIN {X 35.1712,Y -129.1371,Z 161,A -75.6427,B 19.4803,C -0.4323,E1 19.5285,E2 883.8929} C_DIS
LIN {X 38.0995,Y -128.3027,Z 161,A -74.4153,B 19.4803,C -0.4304,E1 19.5318,E2 882.6738} C_DIS
LIN {X 40.8046,Y -127.4671,Z 161,A -73.0246,B 19.4801,C -0.4394,E1 19.5355,E2 881.2596} C_DIS
LIN {X 45.7466,Y -125.7786,Z 161,A -70.9136,B 19.4801,C -0.4368,E1 19.5411,E2 879.162} C_DIS
LIN {X 48.8961,Y -124.5882,Z 161,A -69.5547,B 19.4802,C -0.4352,E1 19.5446,E2 877.812} C_DIS
LIN {X 52.181,Y -123.2494,Z 161,A -67.969,B 19.4802,C -0.4401,E1 19.5487,E2 876.2163} C_DIS
LIN {X 54.9289,Y -122.0482,Z 161,A -66.7149,B 19.4802,C -0.4407,E1 19.5519,E2 874.9645} C_DIS
LIN {X 58.7975,Y -120.2327,Z 161,A -65.0513,B 19.4802,C -0.4364,E1 19.556,E2 873.3196} C_DIS
LIN {X 61.5274,Y -118.8605,Z 161,A -63.6256,B 19.48,C -0.4435,E1 19.5596,E2 871.8778} C_DIS
LIN {X 64.1801,Y -117.4491,Z 161,A -62.1454,B 19.4798,C -0.454,E1 19.5633,E2 870.3718} C_DIS
LIN {X 67.8048,Y -115.3944,Z 161,A -60.4835,B 19.4798,C -0.4518,E1 19.5673,E2 868.723} C_DIS
LIN {X 72.8729,Y -112.2627,Z 161,A -57.9801,B 19.4798,C -0.4544,E1 19.5732,E2 866.2224} C_DIS
LIN {X 76.1238,Y -110.0849,Z 161,A -56.2821,B 19.4798,C -0.4586,E1 19.5771,E2 864.5195} C_DIS
LIN {X 79.53,Y -107.6498,Z 161,A -54.2838,B 19.4794,C -0.4712,E1 19.5817,E2 862.493} C_DIS
LIN {X 83.1153,Y -104.9061,Z 161,A -52.5473,B 19.4795,C -0.4666,E1 19.5855,E2 860.7786} C_DIS
LIN {X 86.2863,Y -102.314,Z 161,A -50.8483,B 19.4795,C -0.468,E1 19.5891,E2 859.084} C_DIS
LIN {X 89.416,Y -99.59,Z 161,A -49.0739,B 19.4795,C -0.4719,E1 19.5928,E2 857.3074} C_DIS
LIN {X 92.7941,Y -96.4503,Z 161,A -47.0538,B 19.4792,C -0.4784,E1 19.597,E2 855.2788} C_DIS
LIN {X 95.9637,Y -93.2975,Z 161,A -45.183,B 19.4792,C -0.4811,E1 19.6006,E2 853.4106} C_DIS
LIN {X 98.8983,Y -90.181,Z 161,A -43.345,B 19.4791,C -0.4857,E1 19.6041,E2 851.5693} C_DIS
LIN {X 102.1732,Y -86.4523,Z 161,A -40.901,B 19.4786,C -0.5052,E1 19.6086,E2 849.082} C_DIS
LIN {X 104.6915,Y -83.385,Z 161,A -39.6615,B 19.479,C -0.4892,E1 19.6107,E2 847.8976} C_DIS
LIN {X 107.0306,Y -80.3612,Z 161,A -37.9534,B 19.4788,C -0.4966,E1 19.6136,E2 846.1782} C_DIS
LIN {X 109.5898,Y -76.8348,Z 161,A -36.0581,B 19.4787,C -0.5029,E1 19.6167,E2 844.2763} C_DIS
LIN {X 113.1312,Y -71.5172,Z 161,A -33.3937,B 19.4785,C -0.5073,E1 19.6208,E2 841.6165} C_DIS
LIN {X 115.2012,Y -68.1338,Z 161,A -31.6843,B 19.4785,C -0.5125,E1 19.6232,E2 839.903} C_DIS
LIN {X 117.8122,Y -63.5114,Z 161,A -29.4052,B 19.4782,C -0.5192,E1 19.6263,E2 837.6196} C_DIS
LIN {X 120.224,Y -58.8152,Z 161,A -27.1543,B 19.4781,C -0.5253,E1 19.6291,E2 835.3661} C_DIS
LIN {X 121.7044,Y -55.6882,Z 161,A -25.7996,B 19.4781,C -0.5241,E1 19.6307,E2 834.0249} C_DIS
LIN {X 122.9205,Y -52.9474,Z 161,A -24.5933,B 19.4781,C -0.5244,E1 19.6321,E2 832.8261} C_DIS
LIN {X 123.9454,Y -50.504,Z 161,A -23.5211,B 19.4781,C -0.525,E1 19.6332,E2 831.7599} C_DIS
LIN {X 125.0936,Y -47.5913,Z 161,A -21.8283,B 19.4776,C -0.5447,E1 19.6349,E2 830.021} C_DIS
LIN {X 126.569,Y -43.5118,Z 161,A -20.1801,B 19.4776,C -0.541,E1 19.6365,E2 828.3959} C_DIS
LIN {X 127.9651,Y -39.2151,Z 161,A -18.4192,B 19.4777,C -0.5392,E1 19.6379,E2 826.6535} C_DIS
LIN {X 128.746,Y -36.5741,Z 161,A -17.0139,B 19.4774,C -0.5529,E1 19.639,E2 825.2181} C_DIS
LIN {X 129.7415,Y -32.8642,Z 161,A -15.5168,B 19.4774,C -0.5514,E1 19.6401,E2 823.7367} C_DIS
LIN {X 130.5933,Y -29.3011,Z 161,A -13.826,B 19.4771,C -0.5617,E1 19.6411,E2 822.0282} C_DIS
LIN {X 131.2985,Y -25.9648,Z 161,A -12.3828,B 19.4771,C -0.5655,E1 19.6419,E2 820.5848} C_DIS
LIN {X 132.1494,Y -21.2138,Z 161,A -10.4928,B 19.4771,C -0.5641,E1 19.6428,E2 818.7135} C_DIS
LIN {X 132.5716,Y -18.3854,Z 161,A -9.2869,B 19.477,C -0.5671,E1 19.6433,E2 817.5079} C_DIS
LIN {X 133.0185,Y -14.8079,Z 161,A -7.7123,B 19.4768,C -0.5734,E1 19.6438,E2 815.9271} C_DIS
LIN {X 133.3555,Y -11.3706,Z 161,A -6.2317,B 19.4767,C -0.5781,E1 19.6442,E2 814.4439} C_DIS
LIN {X 133.6303,Y -7.5121,Z 161,A -4.5007,B 19.4764,C -0.5866,E1 19.6445,E2 812.701} C_DIS
LIN {X 133.8074,Y -3.011,Z 161,A -2.549,B 19.4762,C -0.5937,E1 19.6447,E2 810.7435} C_DIS
LIN {X 133.8359,Y 1.0754,Z 161,A -0.8198,B 19.4761,C -0.5983,E1 19.6447,E2 809.0141} C_DIS
LIN {X 133.7326,Y 5.3483,Z 161,A 0.8439,B 19.4761,C -0.5967,E1 19.6445,E2 807.3683} C_DIS
LIN {X 133.5285,Y 9.1372,Z 161,A 2.5787,B 19.4758,C -0.6067,E1 19.6442,E2 805.6174} C_DIS
LIN {X 133.1603,Y 13.483,Z 161,A 4.4686,B 19.4756,C -0.6135,E1 19.6437,E2 803.7219} C_DIS
LIN {X 132.6956,Y 17.4591,Z 161,A 6.035,B 19.4756,C -0.6123,E1 19.6432,E2 802.1712} C_DIS
LIN {X 132.1871,Y 20.9702,Z 161,A 7.4828,B 19.4756,C -0.6138,E1 19.6426,E2 800.7302} C_DIS
LIN {X 131.6385,Y 24.1789,Z 161,A 9.0356,B 19.4753,C -0.6251,E1 19.6418,E2 799.1556} C_DIS
LIN {X 130.3827,Y 30.2234,Z 161,A 11.5491,B 19.4752,C -0.6274,E1 19.6403,E2 796.6546} C_DIS
LIN {X 129.3342,Y 34.4319,Z 161,A 13.3687,B 19.4751,C -0.6314,E1 19.6391,E2 794.837} C_DIS
LIN {X 128.3174,Y 38.0492,Z 161,A 14.9121,B 19.4751,C -0.6333,E1 19.6379,E2 793.2995} C_DIS
LIN {X 127.3295,Y 41.2356,Z 161,A 16.6779,B 19.4744,C -0.6524,E1 19.6363,E2 791.4901} C_DIS
LIN {X 125.8092,Y 45.6619,Z 161,A 18.3586,B 19.4747,C -0.644,E1 19.6348,E2 789.8468} C_DIS
LIN {X 124.6316,Y 48.7844,Z 161,A 19.7903,B 19.4745,C -0.6482,E1 19.6334,E2 788.413} C_DIS
LIN {X 123.1338,Y 52.4541,Z 161,A 21.4311,B 19.4745,C -0.6505,E1 19.6316,E2 786.7771} C_DIS
LIN {X 122.0074,Y 55.02,Z 161,A 22.675,B 19.4743,C -0.6559,E1 19.6302,E2 785.5263} C_DIS
LIN {X 118.5508,Y 62.1172,Z 161,A 25.8903,B 19.4743,C -0.6579,E1 19.6263,E2 782.3275} C_DIS
LIN {X 117.101,Y 64.8131,Z 161,A 27.4059,B 19.4738,C -0.6703,E1 19.6242,E2 780.7853} C_DIS
LIN {X 114.9383,Y 68.5752,Z 161,A 29.2465,B 19.4737,C -0.6745,E1 19.6216,E2 778.9448} C_DIS
LIN {X 112.5391,Y 72.4461,Z 161,A 31.2246,B 19.4735,C -0.6807,E1 19.6186,E2 776.9612} C_DIS
LIN {X 110.0283,Y 76.2052,Z 161,A 33.1563,B 19.4733,C -0.6854,E1 19.6156,E2 775.0281} C_DIS
LIN {X 107.2513,Y 80.0659,Z 161,A 35.1033,B 19.4733,C -0.6866,E1 19.6124,E2 773.0902} C_DIS
LIN {X 104.6308,Y 83.4612,Z 161,A 36.9862,B 19.473,C -0.6929,E1 19.6091,E2 771.1998} C_DIS
LIN {X 101.728,Y 86.9766,Z 161,A 38.9414,B 19.4729,C -0.6976,E1 19.6056,E2 769.2425} C_DIS
LIN {X 98.7634,Y 90.3287,Z 161,A 40.8288,B 19.4728,C -0.7006,E1 19.6021,E2 767.3571} C_DIS
LIN {X 95.6807,Y 93.5874,Z 161,A 42.7378,B 19.4727,C -0.7043,E1 19.5984,E2 765.4481} C_DIS
LIN {X 92.4068,Y 96.8212,Z 161,A 44.6715,B 19.4726,C -0.7068,E1 19.5945,E2 763.5175} C_DIS
LIN {X 89.2005,Y 99.783,Z 161,A 46.5371,B 19.4724,C -0.7104,E1 19.5907,E2 761.6509} C_DIS
LIN {X 87.0907,Y 101.6302,Z 161,A 47.7449,B 19.4724,C -0.7131,E1 19.5881,E2 760.4415} C_DIS
LIN {X 83.7857,Y 104.3715,Z 161,A 49.6046,B 19.4722,C -0.7174,E1 19.5841,E2 758.5781} C_DIS
LIN {X 80.1882,Y 107.1602,Z 161,A 51.5072,B 19.4722,C -0.7189,E1 19.5799,E2 756.6801} C_DIS
LIN {X 77.0311,Y 109.4513,Z 161,A 53.1103,B 19.4722,C -0.7189,E1 19.5762,E2 755.0844} C_DIS
LIN {X 73.5032,Y 111.851,Z 161,A 54.9154,B 19.4721,C -0.721,E1 19.572,E2 753.2811} C_DIS
LIN {X 70.1884,Y 113.9606,Z 161,A 57.3589,B 19.4708,C -0.756,E1 19.566,E2 750.7433} C_DIS
LIN {X 65.1291,Y 116.9258,Z 161,A 59.0926,B 19.4719,C -0.7265,E1 19.562,E2 749.1045} C_DIS
LIN {X 61.3962,Y 118.9279,Z 161,A 60.8292,B 19.4719,C -0.7257,E1 19.5578,E2 747.3768} C_DIS
LIN {X 57.6487,Y 120.7869,Z 161,A 62.6715,B 19.4717,C -0.7301,E1 19.5531,E2 745.5277} C_DIS
LIN {X 54.4326,Y 122.2702,Z 161,A 64.1949,B 19.4717,C -0.7322,E1 19.5492,E2 744.0031} C_DIS
LIN {X 51.1031,Y 123.6996,Z 161,A 65.6903,B 19.4717,C -0.7315,E1 19.5454,E2 742.5143} C_DIS
LIN {X 48.3386,Y 124.8049,Z 161,A 67.0127,B 19.4716,C -0.7348,E1 19.542,E2 741.1859} C_DIS
LIN {X 45.1808,Y 125.9826,Z 161,A 68.431,B 19.4716,C -0.7352,E1 19.5382,E2 739.7706} C_DIS
LIN {X 41.8923,Y 127.1144,Z 161,A 69.9307,B 19.4715,C -0.7369,E1 19.5343,E2 738.2695} C_DIS
LIN {X 39.0022,Y 128.0302,Z 161,A 71.3009,B 19.4713,C -0.7409,E1 19.5306,E2 736.8905} C_DIS
LIN {X 35.7724,Y 128.9702,Z 161,A 72.6728,B 19.4714,C -0.7392,E1 19.5269,E2 735.527} C_DIS
LIN {X 31.665,Y 130.0397,Z 161,A 74.66,B 19.4711,C -0.7473,E1 19.5215,E2 733.5193} C_DIS
LIN {X 26.7197,Y 131.1449,Z 161,A 76.7172,B 19.4712,C -0.7438,E1 19.5159,E2 731.4761} C_DIS
LIN {X 21.9774,Y 132.0225,Z 161,A 78.7213,B 19.4713,C -0.7422,E1 19.5104,E2 729.4798} C_DIS
LIN {X 18.6321,Y 132.5363,Z 161,A 80.0829,B 19.4714,C -0.7391,E1 19.5067,E2 728.1292} C_DIS
LIN {X 15.4856,Y 132.9409,Z 161,A 81.5732,B 19.4712,C -0.7448,E1 19.5025,E2 726.6232} C_DIS
LIN {X 11.2905,Y 133.3622,Z 161,A 83.3924,B 19.4712,C -0.7456,E1 19.4975,E2 724.8029} C_DIS
LIN {X 7.2768,Y 133.6426,Z 161,A 85.1115,B 19.4712,C -0.7456,E1 19.4927,E2 723.0849} C_DIS
LIN {X 3.7608,Y 133.7866,Z 161,A 86.538,B 19.4713,C -0.7423,E1 19.4887,E2 721.6688} C_DIS
LIN {X -0.3372,Y 133.8396,Z 161,A 88.355,B 19.4713,C -0.7446,E1 19.4836,E2 719.845} C_DIS
LIN {X -4.6291,Y 133.7606,Z 161,A 90.0762,B 19.4714,C -0.7395,E1 19.4789,E2 718.139} C_DIS
LIN {X -8.1248,Y 133.5926,Z 161,A 91.5819,B 19.4714,C -0.7393,E1 19.4747,E2 716.6331} C_DIS
LIN {X -11.3427,Y 133.3578,Z 161,A 93.0026,B 19.4714,C -0.7404,E1 19.4707,E2 715.2085} C_DIS
LIN {X -15.2247,Y 132.972,Z 161,A 94.8087,B 19.4712,C -0.745,E1 19.4656,E2 713.3871} C_DIS
LIN {X -19.2501,Y 132.448,Z 161,A 96.5019,B 19.4713,C -0.7423,E1 19.461,E2 711.7004} C_DIS
LIN {X -23.8844,Y 131.6911,Z 161,A 98.5341,B 19.4713,C -0.7418,E1 19.4554,E2 709.6671} C_DIS
LIN {X -29.2907,Y 130.5957,Z 161,A 100.876,B 19.4714,C -0.7391,E1 19.449,E2 707.3294} C_DIS
LIN {X -32.8521,Y 129.7445,Z 161,A 102.3817,B 19.4716,C -0.7353,E1 19.4449,E2 705.8325} C_DIS
LIN {X -36.7934,Y 128.6847,Z 161,A 104.1672,B 19.4716,C -0.7351,E1 19.4401,E2 704.0439} C_DIS
LIN {X -42.1996,Y 127.0121,Z 161,A 106.3363,B 19.472,C -0.7225,E1 19.4344,E2 701.9076} C_DIS
LIN {X -44.2851,Y 126.3009,Z 161,A 107.4708,B 19.4718,C -0.7289,E1 19.4314,E2 700.7511} C_DIS
LIN {X -47.3498,Y 125.1841,Z 161,A 109.0397,B 19.4716,C -0.734,E1 19.4272,E2 699.1627} C_DIS
LIN {X -51.6822,Y 123.4577,Z 161,A 110.9774,B 19.4718,C -0.7291,E1 19.4222,E2 697.2341} C_DIS
LIN {X -55.859,Y 121.6254,Z 161,A 112.8603,B 19.472,C -0.7236,E1 19.4175,E2 695.3617} C_DIS
LIN {X -59.6106,Y 119.8316,Z 161,A 114.6897,B 19.472,C -0.7228,E1 19.4129,E2 693.5284} C_DIS
LIN {X -63.9537,Y 117.5726,Z 161,A 116.8247,B 19.472,C -0.721,E1 19.4076,E2 691.3911} C_DIS
LIN {X -67.693,Y 115.4601,Z 161,A 118.6999,B 19.4721,C -0.7193,E1 19.403,E2 689.5136} C_DIS
LIN {X -71.6351,Y 113.0568,Z 161,A 120.4968,B 19.4725,C -0.7089,E1 19.3988,E2 687.7407} C_DIS
LIN {X -74.6457,Y 111.0925,Z 161,A 122.1615,B 19.4725,C -0.7109,E1 19.3949,E2 686.0629} C_DIS
LIN {X -77.7264,Y 108.9587,Z 161,A 123.8827,B 19.4724,C -0.7123,E1 19.391,E2 684.3296} C_DIS
LIN {X -81.6022,Y 106.0876,Z 161,A 126.4106,B 19.4719,C -0.726,E1 19.3852,E2 681.7483} C_DIS
LIN {X -85.3059,Y 103.1323,Z 161,A 128.6045,B 19.4719,C -0.7281,E1 19.3805,E2 679.5368} C_DIS
LIN {X -89.5357,Y 99.4828,Z 161,A 130.3466,B 19.4729,C -0.6979,E1 19.377,E2 677.8769} C_DIS
LIN {X -93.8325,Y 95.4392,Z 161,A 132.9998,B 19.4729,C -0.697,E1 19.3717,E2 675.2119} C_DIS
LIN {X -99.8846,Y 89.0871,Z 161,A 136.5582,B 19.4735,C -0.6804,E1 19.3649,E2 671.6829} C_DIS
LIN {X -103.222,Y 85.1976,Z 161,A 138.8647,B 19.4735,C -0.6792,E1 19.3607,E2 669.3661} C_DIS
LIN {X -105.7499,Y 82.0386,Z 161,A 140.6067,B 19.4736,C -0.6752,E1 19.3577,E2 667.6255} C_DIS
LIN {X -108.2231,Y 78.7477,Z 161,A 142.4367,B 19.4737,C -0.6732,E1 19.3547,E2 665.79} C_DIS
LIN {X -110.9275,Y 74.8898,Z 161,A 144.3282,B 19.474,C -0.6631,E1 19.3517,E2 663.9167} C_DIS
LIN {X -113.0576,Y 71.6339,Z 161,A 146.2135,B 19.474,C -0.6668,E1 19.3488,E2 662.0074} C_DIS
LIN {X -115.6216,Y 67.4181,Z 161,A 148.2738,B 19.4742,C -0.659,E1 19.3459,E2 659.9567} C_DIS
LIN {X -117.7289,Y 63.6664,Z 161,A 150.0726,B 19.4744,C -0.6522,E1 19.3435,E2 658.166} C_DIS
LIN {X -121.6056,Y 55.9018,Z 161,A 153.6569,B 19.4749,C -0.6365,E1 19.3391,E2 654.6035} C_DIS
LIN {X -123.7485,Y 50.9859,Z 161,A 156.0235,B 19.475,C -0.6324,E1 19.3365,E2 652.2321} C_DIS
LIN {X -124.8061,Y 48.3356,Z 161,A 157.3611,B 19.475,C -0.6331,E1 19.3351,E2 650.8824} C_DIS
LIN {X -126.0065,Y 45.1145,Z 161,A 158.7381,B 19.4753,C -0.6252,E1 19.3338,E2 649.5192} C_DIS
LIN {X -127.0769,Y 42.0051,Z 161,A 160.4847,B 19.475,C -0.6336,E1 19.3322,E2 647.7339} C_DIS
LIN {X -128.5095,Y 37.3931,Z 161,A 162.5065,B 19.4752,C -0.6256,E1 19.3306,E2 645.7209} C_DIS
LIN {X -129.9591,Y 31.9995,Z 161,A 165.2552,B 19.4751,C -0.6316,E1 19.3287,E2 642.9326} C_DIS
LIN {X -130.9877,Y 27.4907,Z 161,A 166.6748,B 19.4759,C -0.6045,E1 19.3279,E2 641.5843} C_DIS
LIN {X -132.0284,Y 21.9415,Z 161,A 169.1375,B 19.4761,C -0.5986,E1 19.3267,E2 639.1199} C_DIS
LIN {X -132.5153,Y 18.779,Z 161,A 170.5244,B 19.4761,C -0.595,E1 19.3261,E2 637.733} C_DIS
LIN {X -133.056,Y 14.4594,Z 161,A 172.3003,B 19.4764,C -0.5859,E1 19.3256,E2 635.9706} C_DIS
LIN {X -133.3066,Y 11.9492,Z 161,A 173.4206,B 19.4764,C -0.584,E1 19.3253,E2 634.8472} C_DIS
LIN {X -133.5743,Y 8.4215,Z 161,A 175.0154,B 19.4765,C -0.5823,E1 19.3249,E2 633.245} C_DIS
LIN {X -133.7415,Y 5.1187,Z 161,A 176.4577,B 19.4766,C -0.5788,E1 19.3248,E2 631.8016} C_DIS
LIN {X -133.8361,Y 1.0473,Z 161,A 178.2742,B 19.4767,C -0.5761,E1 19.3247,E2 629.979} C_DIS
LIN {X -133.8132,Y -2.6915,Z 161,A 179.9225,B 19.4768,C -0.5728,E1 19.3247,E2 628.3273} C_DIS
LIN {X -133.6748,Y -6.6366,Z 161,A -178.4822,B 19.477,C -0.564,E1 19.3249,E2 626.7459} C_DIS
LIN {X -133.4582,Y -10.0999,Z 161,A -176.852,B 19.477,C -0.5648,E1 19.3253,E2 625.1005} C_DIS
LIN {X -133.1512,Y -13.575,Z 161,A -175.5198,B 19.4773,C -0.5541,E1 19.3256,E2 623.79} C_DIS
LIN {X -132.668,Y -17.6701,Z 161,A -173.7144,B 19.4774,C -0.5502,E1 19.3262,E2 621.9822} C_DIS
LIN {X -132.1625,Y -21.1294,Z 161,A -171.9791,B 19.4774,C -0.5545,E1 19.327,E2 620.2202} C_DIS
LIN {X -131.3629,Y -25.6312,Z 161,A -170.1688,B 19.4776,C -0.543,E1 19.3279,E2 618.4304} C_DIS
LIN {X -129.9528,Y -32.0254,Z 161,A -167.2681,B 19.4777,C -0.5382,E1 19.3297,E2 615.5218} C_DIS
LIN {X -128.9064,Y -36.0004,Z 161,A -165.5189,B 19.4779,C -0.5326,E1 19.331,E2 613.7762} C_DIS
LIN {X -127.837,Y -39.6337,Z 161,A -164.0098,B 19.4781,C -0.5236,E1 19.3322,E2 612.2829} C_DIS
LIN {X -126.8882,Y -42.5718,Z 161,A -162.683,B 19.4782,C -0.5199,E1 19.3334,E2 610.9572} C_DIS
LIN {X -125.7996,Y -45.6883,Z 161,A -161.2105,B 19.4782,C -0.5181,E1 19.3348,E2 609.4792} C_DIS
LIN {X -124.6234,Y -48.8056,Z 161,A -159.7965,B 19.4784,C -0.5135,E1 19.3362,E2 608.0685} C_DIS
LIN {X -123.2811,Y -52.1052,Z 161,A -158.1075,B 19.4784,C -0.5154,E1 19.338,E2 606.3613} C_DIS
LIN {X -121.776,Y -55.5334,Z 161,A -156.6646,B 19.4786,C -0.5048,E1 19.3396,E2 604.9399} C_DIS
LIN {X -119.7077,Y -59.8619,Z 161,A -154.5762,B 19.4787,C -0.5005,E1 19.3422,E2 602.8497} C_DIS
LIN {X -118.0797,Y -63.0135,Z 161,A -152.9065,B 19.4787,C -0.5022,E1 19.3444,E2 601.1633} C_DIS
LIN {X -115.9229,Y -66.8976,Z 161,A -151.0449,B 19.4788,C -0.4956,E1 19.3469,E2 599.3086} C_DIS
LIN {X -113.7244,Y -70.5702,Z 161,A -148.9393,B 19.4787,C -0.5014,E1 19.3501,E2 597.1714} C_DIS
LIN {X -111.8584,Y -73.492,Z 161,A -147.8308,B 19.4791,C -0.4832,E1 19.3517,E2 596.1103} C_DIS
LIN {X -109.5815,Y -76.8465,Z 161,A -145.9123,B 19.4791,C -0.4859,E1 19.3547,E2 594.1712} C_DIS
LIN {X -106.9509,Y -80.4668,Z 161,A -143.9948,B 19.4791,C -0.4813,E1 19.3579,E2 592.2553} C_DIS
LIN {X -104.3187,Y -83.8512,Z 161,A -142.1925,B 19.4793,C -0.4758,E1 19.361,E2 590.4587} C_DIS
LIN {X -101.6122,Y -87.1116,Z 161,A -140.3056,B 19.4793,C -0.4744,E1 19.3645,E2 588.5643} C_DIS
LIN {X -99.037,Y -90.0281,Z 161,A -138.6803,B 19.4795,C -0.4692,E1 19.3675,E2 586.9454} C_DIS
LIN {X -96.0438,Y -93.2147,Z 161,A -136.7791,B 19.4795,C -0.4663,E1 19.3712,E2 585.0419} C_DIS
LIN {X -92.825,Y -96.4211,Z 161,A -134.7939,B 19.4795,C -0.4639,E1 19.3751,E2 583.0532} C_DIS
LIN {X -89.6236,Y -99.4039,Z 161,A -132.961,B 19.4797,C -0.4586,E1 19.3789,E2 581.2265} C_DIS
LIN {X -86.5761,Y -102.0684,Z 161,A -131.0909,B 19.4797,C -0.4607,E1 19.3829,E2 579.3406} C_DIS
LIN {X -83.4315,Y -104.6545,Z 161,A -129.4543,B 19.4798,C -0.4533,E1 19.3864,E2 577.718} C_DIS
LIN {X -79.9375,Y -107.3469,Z 161,A -127.5642,B 19.4798,C -0.4501,E1 19.3906,E2 575.8287} C_DIS
LIN {X -76.3255,Y -109.9445,Z 161,A -125.8403,B 19.4801,C -0.4398,E1 19.3945,E2 574.1279} C_DIS
LIN {X -73.4513,Y -111.8852,Z 161,A -124.1695,B 19.4801,C -0.4448,E1 19.3984,E2 572.4349} C_DIS
LIN {X -70.2061,Y -113.9497,Z 161,A -122.4797,B 19.4801,C -0.444,E1 19.4024,E2 570.7404} C_DIS
LIN {X -66.259,Y -116.2889,Z 161,A -120.5643,B 19.4801,C -0.4393,E1 19.407,E2 568.8317} C_DIS
LIN {X -62.6246,Y -118.2844,Z 161,A -118.7205,B 19.4801,C -0.4397,E1 19.4116,E2 566.9798} C_DIS
LIN {X -58.9528,Y -120.1561,Z 161,A -117.0727,B 19.4803,C -0.4328,E1 19.4157,E2 565.3468} C_DIS
LIN {X -55.8621,Y -121.6239,Z 161,A -115.5864,B 19.4803,C -0.432,E1 19.4194,E2 563.8581} C_DIS
LIN {X -52.899,Y -122.9415,Z 161,A -114.2579,B 19.4803,C -0.4281,E1 19.4228,E2 562.5372} C_DIS
LIN {X -50.0578,Y -124.1252,Z 161,A -112.885,B 19.4803,C -0.429,E1 19.4264,E2 561.1577} C_DIS
LIN {X -46.9195,Y -125.3452,Z 161,A -111.4598,B 19.4803,C -0.427,E1 19.4301,E2 559.7346} C_DIS
LIN {X -43.2999,Y -126.6425,Z 161,A -109.8528,B 19.4805,C -0.424,E1 19.4343,E2 558.1325} C_DIS
LIN {X -40.0742,Y -127.7004,Z 161,A -108.363,B 19.4805,C -0.4243,E1 19.4383,E2 556.6381} C_DIS
LIN {X -37.1874,Y -128.5697,Z 161,A -107.0345,B 19.4805,C -0.4249,E1 19.4419,E2 555.3049} C_DIS
LIN {X -32.2015,Y -129.9097,Z 161,A -104.8566,B 19.4805,C -0.4222,E1 19.4477,E2 553.1308} C_DIS
LIN {X -28.1766,Y -130.8396,Z 161,A -103.0562,B 19.4805,C -0.4227,E1 19.4527,E2 551.3262} C_DIS
LIN {X -24.2758,Y -131.6211,Z 161,A -101.405,B 19.4805,C -0.4198,E1 19.4572,E2 549.6812} C_DIS
LIN {X -20.7551,Y -132.2204,Z 161,A -99.795,B 19.4805,C -0.4227,E1 19.4616,E2 548.0607} C_DIS
LIN {X -17.3183,Y -132.7141,Z 161,A -98.3286,B 19.4805,C -0.4215,E1 19.4657,E2 546.5963} C_DIS
LIN {X -13.4641,Y -133.1621,Z 161,A -96.5404,B 19.4805,C -0.4264,E1 19.4707,E2 544.7918} C_DIS
Enddeposition()
END
